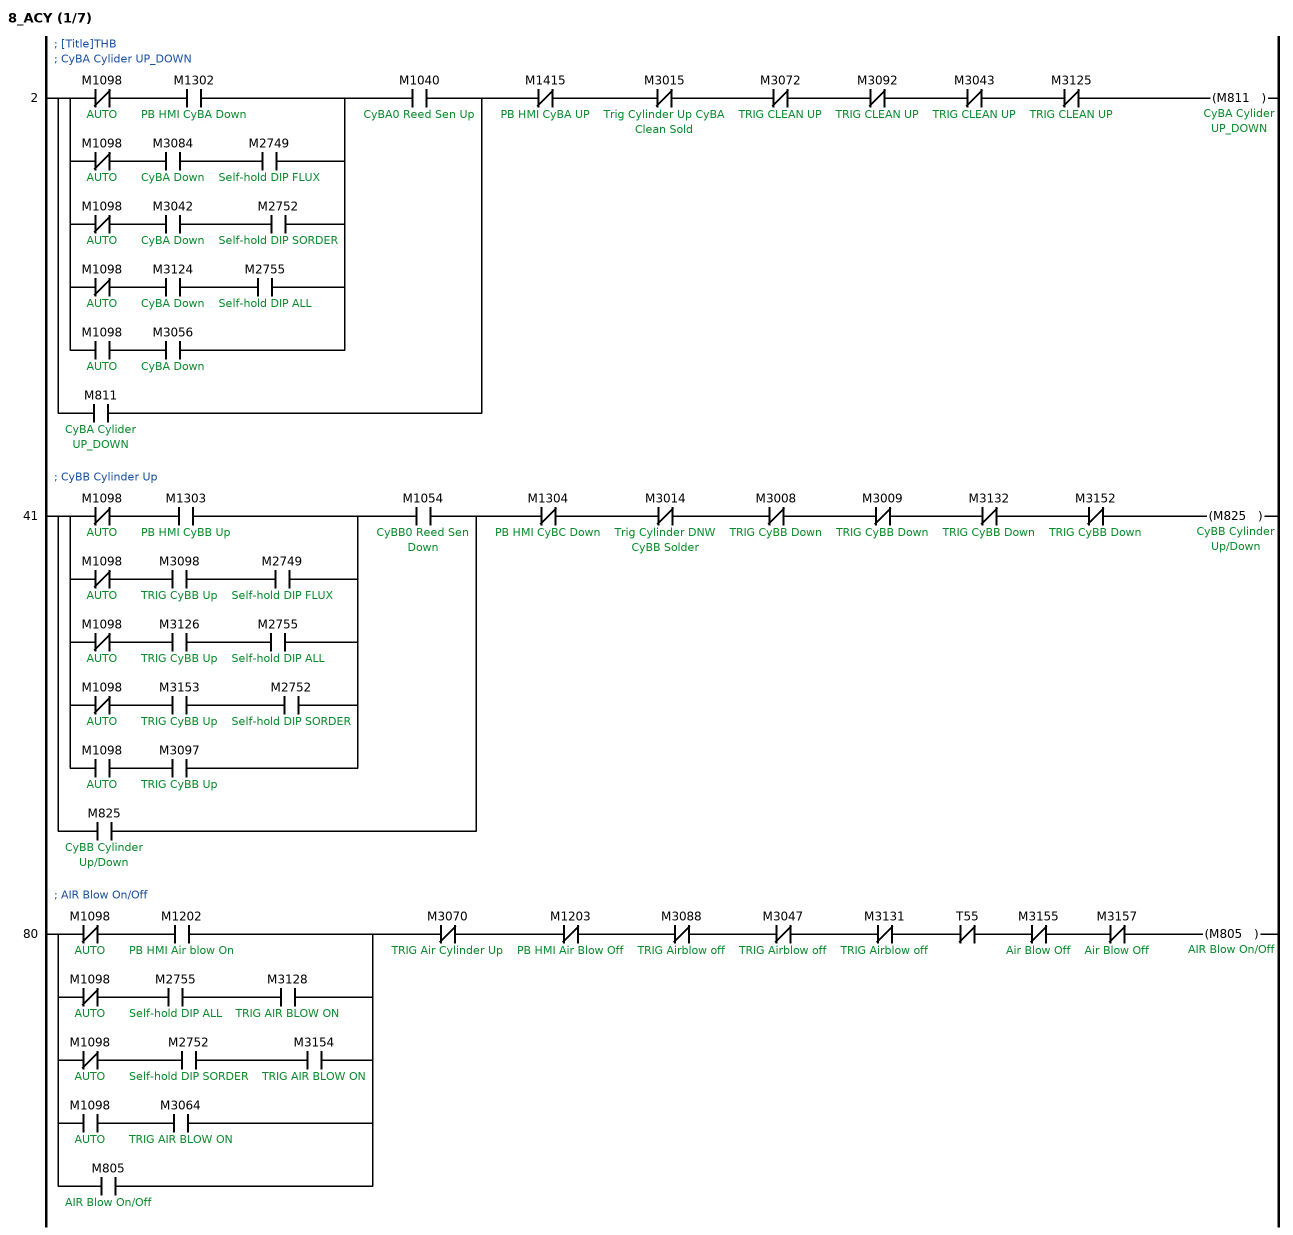
[picture p96: ladder of 8_ACY, rungs at steps 2 to 80]
; [Title]THB
; CyBA Cylider UP_DOWN
2     LDI     M1098  ; AUTO
      AND     M1302  ; PB HMI CyBA Down
      LDI     M1098  ; AUTO
      AND     M3084  ; CyBA Down
      AND     M2749  ; Self-hold DIP FLUX
      ORB
      LDI     M1098  ; AUTO
      AND     M3042  ; CyBA Down
      AND     M2752  ; Self-hold DIP SORDER
      ORB
      LDI     M1098  ; AUTO
      AND     M3124  ; CyBA Down
      AND     M2755  ; Self-hold DIP ALL
      ORB
      LD      M1098  ; AUTO
      AND     M3056  ; CyBA Down
      ORB
      AND     M1040  ; CyBA0 Reed Sen Up
      OR      M811  ; CyBA Cylider UP_DOWN
      ANI     M1415  ; PB HMI CyBA UP
      ANI     M3015  ; Trig Cylinder Up CyBA Clean Sold
      ANI     M3072  ; TRIG CLEAN UP
      ANI     M3092  ; TRIG CLEAN UP
      ANI     M3043  ; TRIG CLEAN UP
      ANI     M3125  ; TRIG CLEAN UP
      OUT     M811  ; CyBA Cylider UP_DOWN
; CyBB Cylinder Up
41    LDI     M1098  ; AUTO
      AND     M1303  ; PB HMI CyBB Up
      LDI     M1098  ; AUTO
      AND     M3098  ; TRIG CyBB Up
      AND     M2749  ; Self-hold DIP FLUX
      ORB
      LDI     M1098  ; AUTO
      AND     M3126  ; TRIG CyBB Up
      AND     M2755  ; Self-hold DIP ALL
      ORB
      LDI     M1098  ; AUTO
      AND     M3153  ; TRIG CyBB Up
      AND     M2752  ; Self-hold DIP SORDER
      ORB
      LD      M1098  ; AUTO
      AND     M3097  ; TRIG CyBB Up
      ORB
      AND     M1054  ; CyBB0 Reed Sen Down
      OR      M825  ; CyBB Cylinder Up/Down
      ANI     M1304  ; PB HMI CyBC Down
      ANI     M3014  ; Trig Cylinder DNW CyBB Solder
      ANI     M3008  ; TRIG CyBB Down
      ANI     M3009  ; TRIG CyBB Down
      ANI     M3132  ; TRIG CyBB Down
      ANI     M3152  ; TRIG CyBB Down
      OUT     M825  ; CyBB Cylinder Up/Down
; AIR Blow On/Off
80    LDI     M1098  ; AUTO
      AND     M1202  ; PB HMI Air blow On
      LDI     M1098  ; AUTO
      AND     M2755  ; Self-hold DIP ALL
      AND     M3128  ; TRIG AIR BLOW ON
      ORB
      LDI     M1098  ; AUTO
      AND     M2752  ; Self-hold DIP SORDER
      AND     M3154  ; TRIG AIR BLOW ON
      ORB
      LD      M1098  ; AUTO
      AND     M3064  ; TRIG AIR BLOW ON
      ORB
      OR      M805  ; AIR Blow On/Off
      ANI     M3070  ; TRIG Air Cylinder Up
      ANI     M1203  ; PB HMI Air Blow Off
      ANI     M3088  ; TRIG Airblow off
      ANI     M3047  ; TRIG Airblow off
      ANI     M3131  ; TRIG Airblow off
      ANI     T55
      ANI     M3155  ; Air Blow Off
      ANI     M3157  ; Air Blow Off
      OUT     M805  ; AIR Blow On/Off
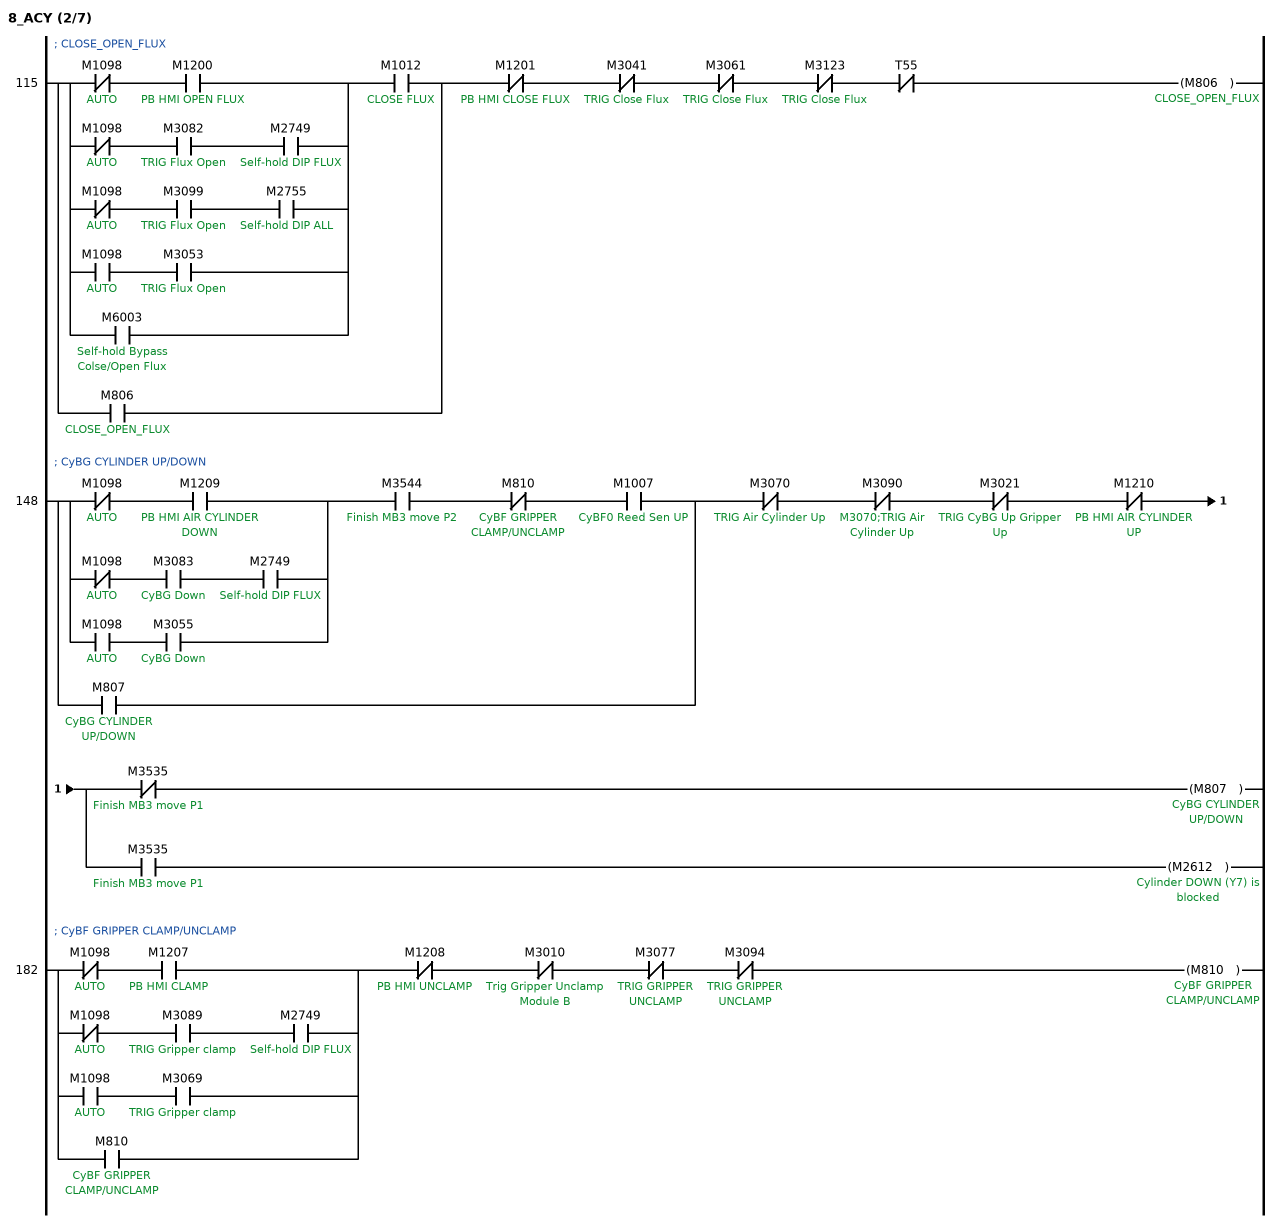
; CLOSE_OPEN_FLUX
115   LDI     M1098  ; AUTO
      AND     M1200  ; PB HMI OPEN FLUX
      LDI     M1098  ; AUTO
      AND     M3082  ; TRIG Flux Open
      AND     M2749  ; Self-hold DIP FLUX
      ORB
      LDI     M1098  ; AUTO
      AND     M3099  ; TRIG Flux Open
      AND     M2755  ; Self-hold DIP ALL
      ORB
      LD      M1098  ; AUTO
      AND     M3053  ; TRIG Flux Open
      ORB
      OR      M6003  ; Self-hold Bypass Colse/Open Flux
      AND     M1012  ; CLOSE FLUX
      OR      M806  ; CLOSE_OPEN_FLUX
      ANI     M1201  ; PB HMI CLOSE FLUX
      ANI     M3041  ; TRIG Close Flux
      ANI     M3061  ; TRIG Close Flux
      ANI     M3123  ; TRIG Close Flux
      ANI     T55
      OUT     M806  ; CLOSE_OPEN_FLUX
; CyBG CYLINDER UP/DOWN
148   LDI     M1098  ; AUTO
      AND     M1209  ; PB HMI AIR CYLINDER DOWN
      LDI     M1098  ; AUTO
      AND     M3083  ; CyBG Down
      AND     M2749  ; Self-hold DIP FLUX
      ORB
      LD      M1098  ; AUTO
      AND     M3055  ; CyBG Down
      ORB
      AND     M3544  ; Finish MB3 move P2
      ANI     M810  ; CyBF GRIPPER CLAMP/UNCLAMP
      AND     M1007  ; CyBF0 Reed Sen UP
      OR      M807  ; CyBG CYLINDER UP/DOWN
      ANI     M3070  ; TRIG Air Cylinder Up
      ANI     M3090  ; M3070;TRIG Air Cylinder Up
      ANI     M3021  ; TRIG CyBG Up Gripper Up
      ANI     M1210  ; PB HMI AIR CYLINDER UP
      MPS
      ANI     M3535  ; Finish MB3 move P1
      OUT     M807  ; CyBG CYLINDER UP/DOWN
      MPP
      AND     M3535  ; Finish MB3 move P1
      OUT     M2612  ; Cylinder DOWN (Y7) is blocked
; CyBF GRIPPER CLAMP/UNCLAMP
182   LDI     M1098  ; AUTO
      AND     M1207  ; PB HMI CLAMP
      LDI     M1098  ; AUTO
      AND     M3089  ; TRIG Gripper clamp
      AND     M2749  ; Self-hold DIP FLUX
      ORB
      LD      M1098  ; AUTO
      AND     M3069  ; TRIG Gripper clamp
      ORB
      OR      M810  ; CyBF GRIPPER CLAMP/UNCLAMP
      ANI     M1208  ; PB HMI UNCLAMP
      ANI     M3010  ; Trig Gripper Unclamp Module B
      ANI     M3077  ; TRIG GRIPPER UNCLAMP
      ANI     M3094  ; TRIG GRIPPER UNCLAMP
      OUT     M810  ; CyBF GRIPPER CLAMP/UNCLAMP
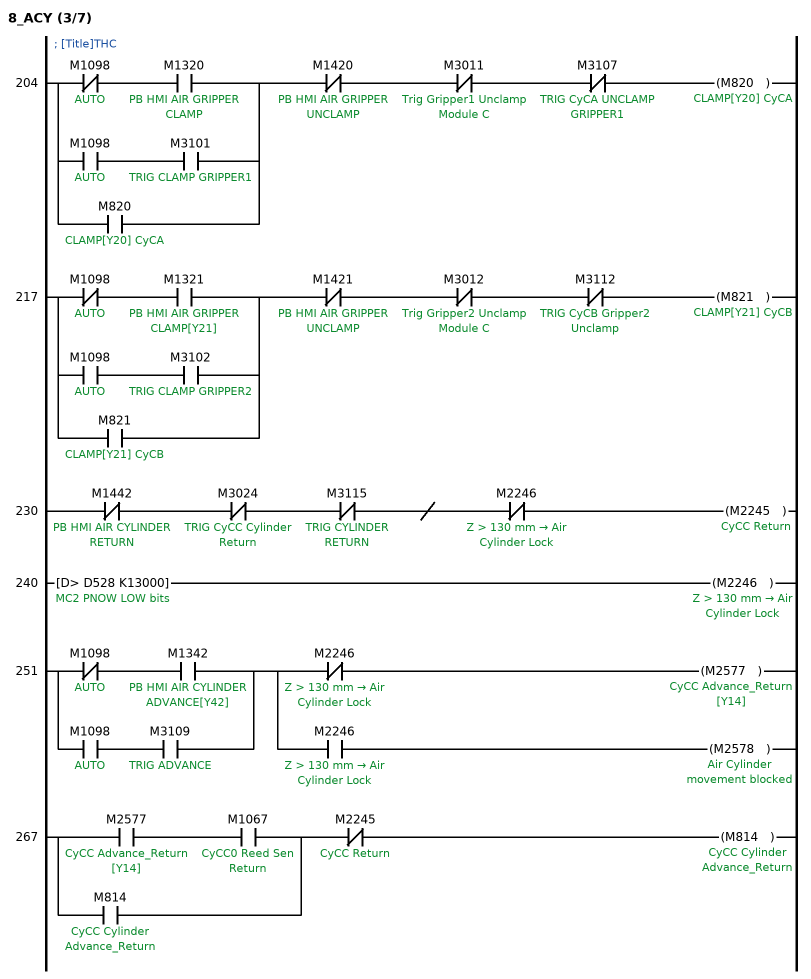
; [Title]THC
204   LDI     M1098  ; AUTO
      AND     M1320  ; PB HMI AIR GRIPPER CLAMP
      LD      M1098  ; AUTO
      AND     M3101  ; TRIG CLAMP GRIPPER1
      ORB
      OR      M820  ; CLAMP[Y20] CyCA
      ANI     M1420  ; PB HMI AIR GRIPPER UNCLAMP
      ANI     M3011  ; Trig Gripper1 Unclamp Module C
      ANI     M3107  ; TRIG CyCA UNCLAMP GRIPPER1
      OUT     M820  ; CLAMP[Y20] CyCA
217   LDI     M1098  ; AUTO
      AND     M1321  ; PB HMI AIR GRIPPER CLAMP[Y21]
      LD      M1098  ; AUTO
      AND     M3102  ; TRIG CLAMP GRIPPER2
      ORB
      OR      M821  ; CLAMP[Y21] CyCB
      ANI     M1421  ; PB HMI AIR GRIPPER UNCLAMP
      ANI     M3012  ; Trig Gripper2 Unclamp Module C
      ANI     M3112  ; TRIG CyCB Gripper2 Unclamp
      OUT     M821  ; CLAMP[Y21] CyCB
230   LDI     M1442  ; PB HMI AIR CYLINDER RETURN
      ANI     M3024  ; TRIG CyCC Cylinder Return
      ANI     M3115  ; TRIG CYLINDER RETURN
      INV
      ANI     M2246  ; Z > 130 mm → Air Cylinder Lock
      OUT     M2245  ; CyCC Return
240   LDD>    D528 K13000  ; MC2 PNOW LOW bits
      OUT     M2246  ; Z > 130 mm → Air Cylinder Lock
251   LDI     M1098  ; AUTO
      AND     M1342  ; PB HMI AIR CYLINDER ADVANCE[Y42]
      LD      M1098  ; AUTO
      AND     M3109  ; TRIG ADVANCE
      ORB
      MPS
      ANI     M2246  ; Z > 130 mm → Air Cylinder Lock
      OUT     M2577  ; CyCC Advance_Return [Y14]
      MPP
      AND     M2246  ; Z > 130 mm → Air Cylinder Lock
      OUT     M2578  ; Air Cylinder movement blocked
267   LD      M2577  ; CyCC Advance_Return [Y14]
      AND     M1067  ; CyCC0 Reed Sen Return
      OR      M814  ; CyCC Cylinder Advance_Return
      ANI     M2245  ; CyCC Return
      OUT     M814  ; CyCC Cylinder Advance_Return
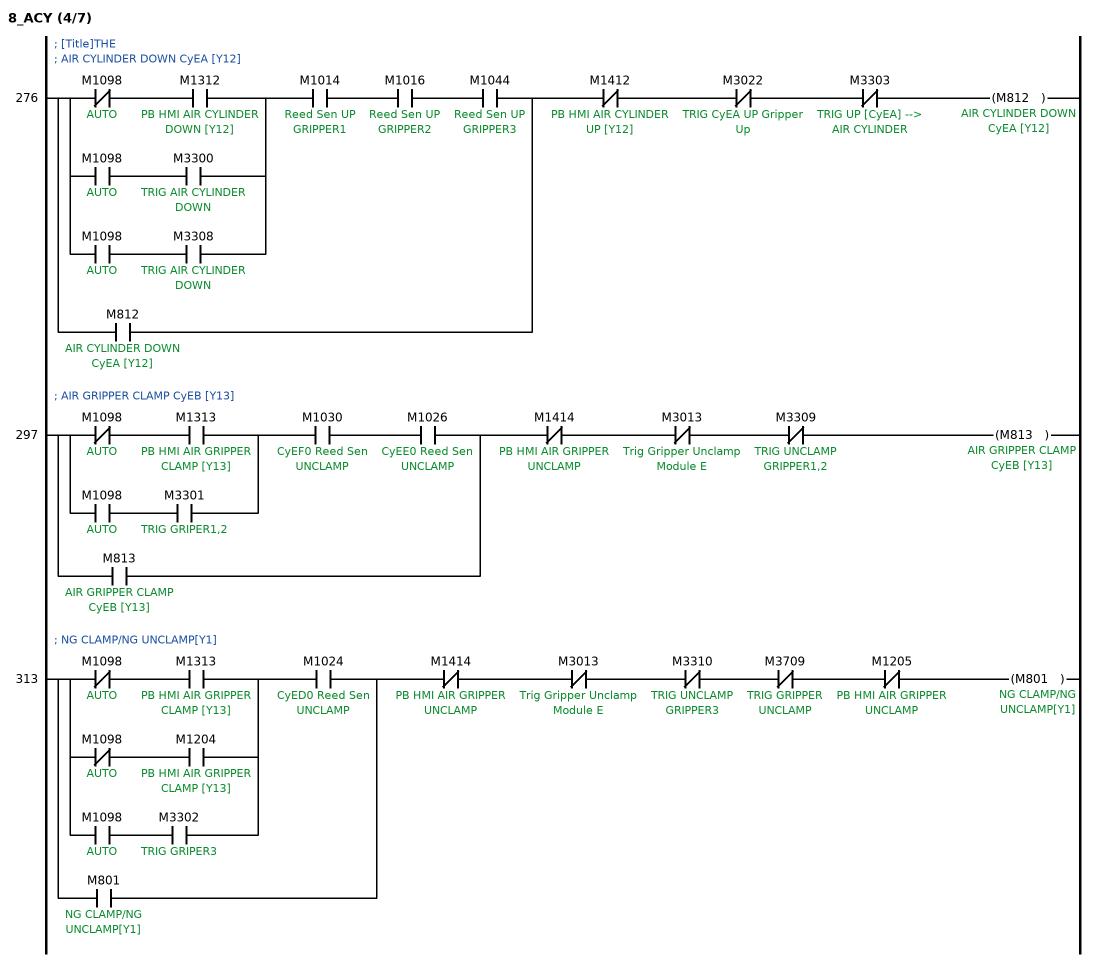
; [Title]THE
; AIR CYLINDER DOWN CyEA [Y12]
276   LDI     M1098  ; AUTO
      AND     M1312  ; PB HMI AIR CYLINDER DOWN [Y12]
      LD      M1098  ; AUTO
      AND     M3300  ; TRIG AIR CYLINDER DOWN
      ORB
      LD      M1098  ; AUTO
      AND     M3308  ; TRIG AIR CYLINDER DOWN
      ORB
      AND     M1014  ; Reed Sen UP GRIPPER1
      AND     M1016  ; Reed Sen UP GRIPPER2
      AND     M1044  ; Reed Sen UP GRIPPER3
      OR      M812  ; AIR CYLINDER DOWN CyEA [Y12]
      ANI     M1412  ; PB HMI AIR CYLINDER UP [Y12]
      ANI     M3022  ; TRIG CyEA UP Gripper Up
      ANI     M3303  ; TRIG UP [CyEA] --> AIR CYLINDER
      OUT     M812  ; AIR CYLINDER DOWN CyEA [Y12]
; AIR GRIPPER CLAMP CyEB [Y13]
297   LDI     M1098  ; AUTO
      AND     M1313  ; PB HMI AIR GRIPPER CLAMP [Y13]
      LD      M1098  ; AUTO
      AND     M3301  ; TRIG GRIPER1,2
      ORB
      AND     M1030  ; CyEF0 Reed Sen UNCLAMP
      AND     M1026  ; CyEE0 Reed Sen UNCLAMP
      OR      M813  ; AIR GRIPPER CLAMP CyEB [Y13]
      ANI     M1414  ; PB HMI AIR GRIPPER UNCLAMP
      ANI     M3013  ; Trig Gripper Unclamp Module E
      ANI     M3309  ; TRIG UNCLAMP GRIPPER1,2
      OUT     M813  ; AIR GRIPPER CLAMP CyEB [Y13]
; NG CLAMP/NG UNCLAMP[Y1]
313   LDI     M1098  ; AUTO
      AND     M1313  ; PB HMI AIR GRIPPER CLAMP [Y13]
      LDI     M1098  ; AUTO
      AND     M1204  ; PB HMI AIR GRIPPER CLAMP [Y13]
      ORB
      LD      M1098  ; AUTO
      AND     M3302  ; TRIG GRIPER3
      ORB
      AND     M1024  ; CyED0 Reed Sen UNCLAMP
      OR      M801  ; NG CLAMP/NG UNCLAMP[Y1]
      ANI     M1414  ; PB HMI AIR GRIPPER UNCLAMP
      ANI     M3013  ; Trig Gripper Unclamp Module E
      ANI     M3310  ; TRIG UNCLAMP GRIPPER3
      ANI     M3709  ; TRIG GRIPPER UNCLAMP
      ANI     M1205  ; PB HMI AIR GRIPPER UNCLAMP
      OUT     M801  ; NG CLAMP/NG UNCLAMP[Y1]
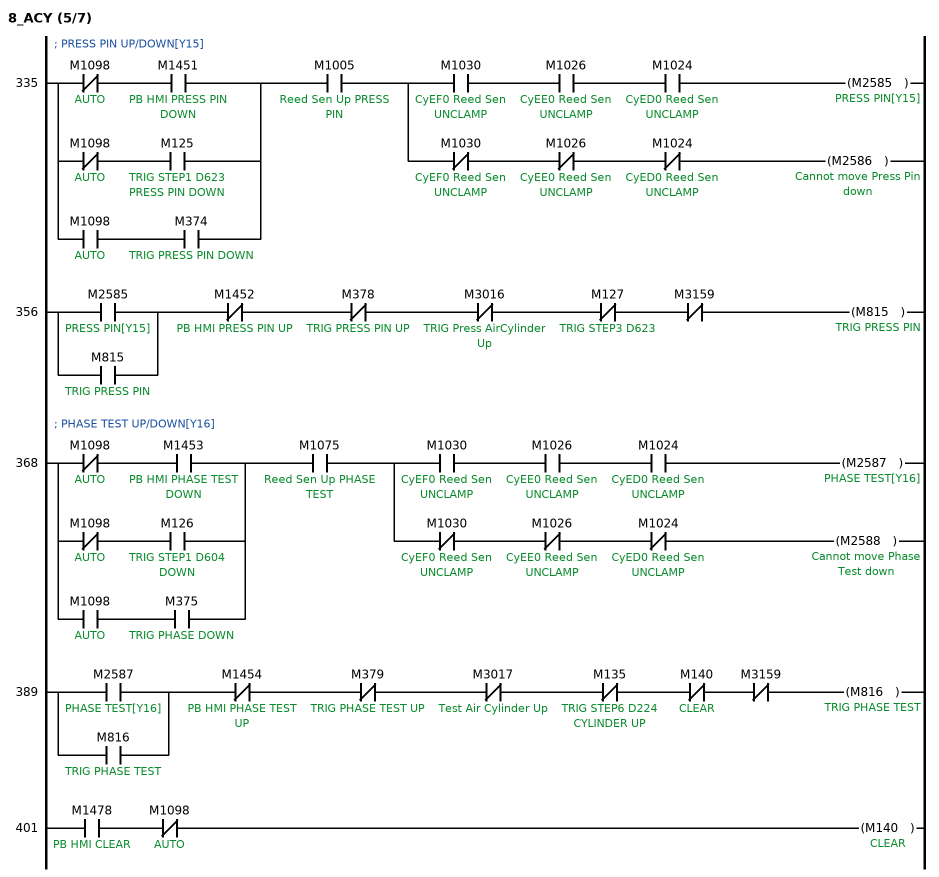
; PRESS PIN UP/DOWN[Y15]
335   LDI     M1098  ; AUTO
      AND     M1451  ; PB HMI PRESS PIN DOWN
      LDI     M1098  ; AUTO
      AND     M125  ; TRIG STEP1 D623 PRESS PIN DOWN
      ORB
      LD      M1098  ; AUTO
      AND     M374  ; TRIG PRESS PIN DOWN
      ORB
      AND     M1005  ; Reed Sen Up PRESS PIN
      MPS
      AND     M1030  ; CyEF0 Reed Sen UNCLAMP
      AND     M1026  ; CyEE0 Reed Sen UNCLAMP
      AND     M1024  ; CyED0 Reed Sen UNCLAMP
      OUT     M2585  ; PRESS PIN[Y15]
      MPP
      ANI     M1030  ; CyEF0 Reed Sen UNCLAMP
      ANI     M1026  ; CyEE0 Reed Sen UNCLAMP
      ANI     M1024  ; CyED0 Reed Sen UNCLAMP
      OUT     M2586  ; Cannot move Press Pin down
356   LD      M2585  ; PRESS PIN[Y15]
      OR      M815  ; TRIG PRESS PIN
      ANI     M1452  ; PB HMI PRESS PIN UP
      ANI     M378  ; TRIG PRESS PIN UP
      ANI     M3016  ; TRIG Press AirCylinder Up
      ANI     M127  ; TRIG STEP3 D623
      ANI     M3159
      OUT     M815  ; TRIG PRESS PIN
; PHASE TEST UP/DOWN[Y16]
368   LDI     M1098  ; AUTO
      AND     M1453  ; PB HMI PHASE TEST DOWN
      LDI     M1098  ; AUTO
      AND     M126  ; TRIG STEP1 D604 DOWN
      ORB
      LD      M1098  ; AUTO
      AND     M375  ; TRIG PHASE DOWN
      ORB
      AND     M1075  ; Reed Sen Up PHASE TEST
      MPS
      AND     M1030  ; CyEF0 Reed Sen UNCLAMP
      AND     M1026  ; CyEE0 Reed Sen UNCLAMP
      AND     M1024  ; CyED0 Reed Sen UNCLAMP
      OUT     M2587  ; PHASE TEST[Y16]
      MPP
      ANI     M1030  ; CyEF0 Reed Sen UNCLAMP
      ANI     M1026  ; CyEE0 Reed Sen UNCLAMP
      ANI     M1024  ; CyED0 Reed Sen UNCLAMP
      OUT     M2588  ; Cannot move Phase Test down
389   LD      M2587  ; PHASE TEST[Y16]
      OR      M816  ; TRIG PHASE TEST
      ANI     M1454  ; PB HMI PHASE TEST UP
      ANI     M379  ; TRIG PHASE TEST UP
      ANI     M3017  ; Test Air Cylinder Up
      ANI     M135  ; TRIG STEP6 D224 CYLINDER UP
      ANI     M140  ; CLEAR
      ANI     M3159
      OUT     M816  ; TRIG PHASE TEST
401   LD      M1478  ; PB HMI CLEAR
      ANI     M1098  ; AUTO
      OUT     M140  ; CLEAR
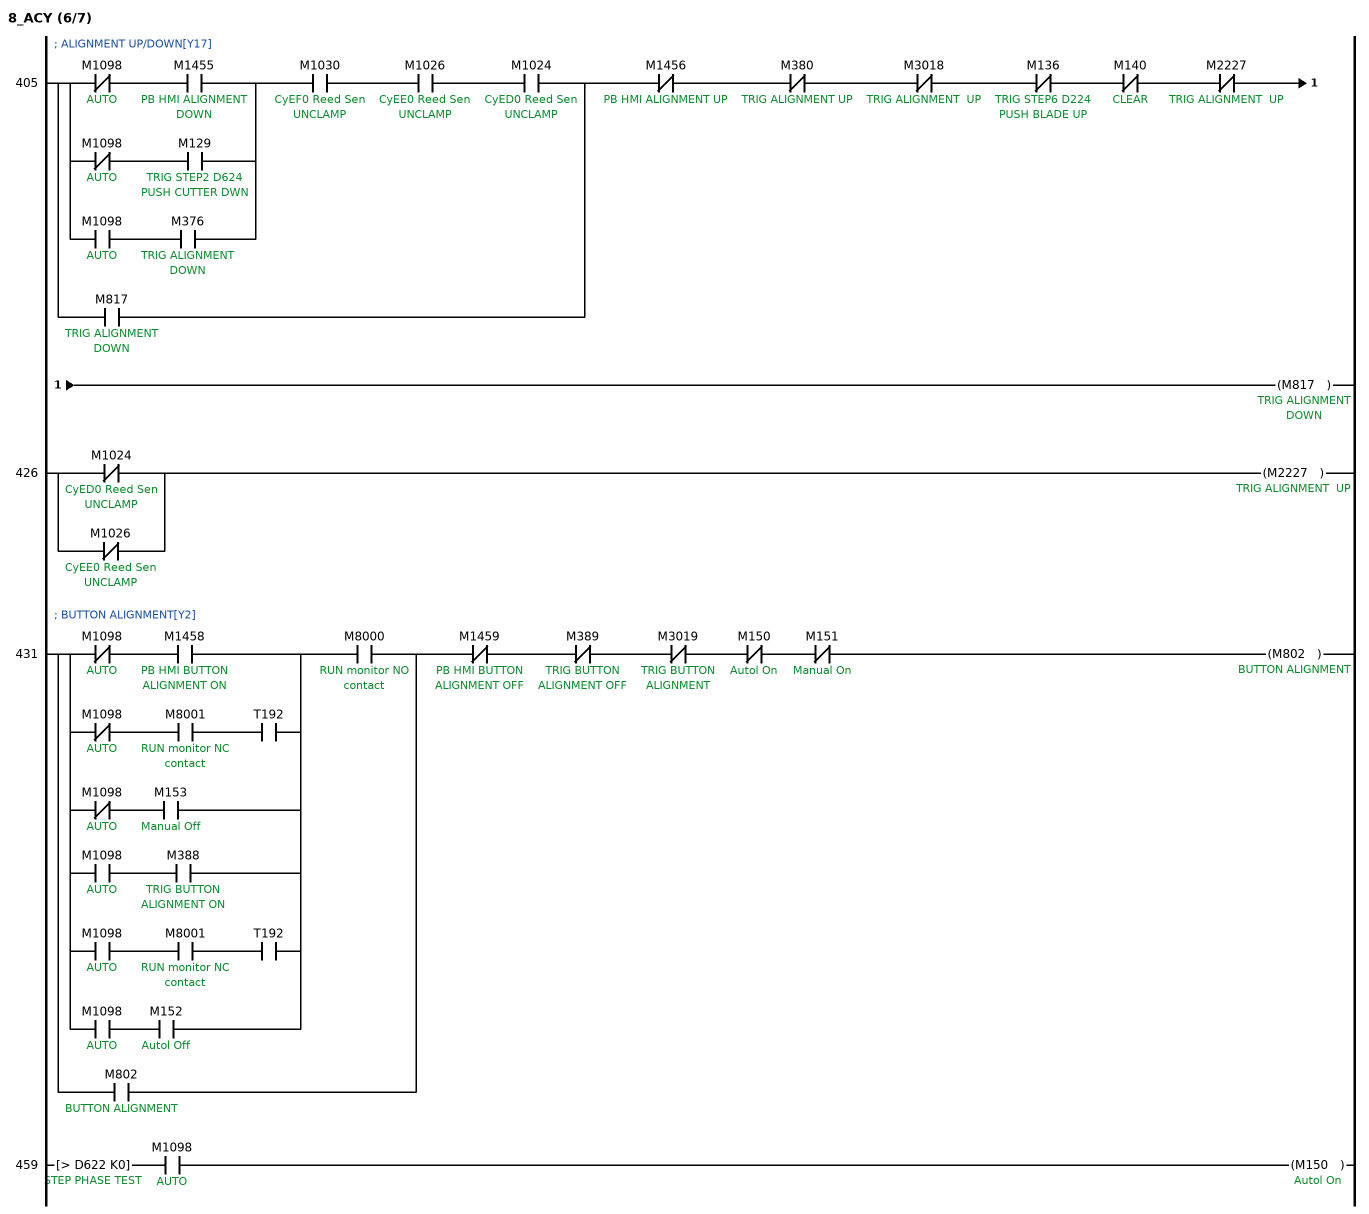
; ALIGNMENT UP/DOWN[Y17]
405   LDI     M1098  ; AUTO
      AND     M1455  ; PB HMI ALIGNMENT DOWN
      LDI     M1098  ; AUTO
      AND     M129  ; TRIG STEP2 D624 PUSH CUTTER DWN
      ORB
      LD      M1098  ; AUTO
      AND     M376  ; TRIG ALIGNMENT DOWN
      ORB
      AND     M1030  ; CyEF0 Reed Sen UNCLAMP
      AND     M1026  ; CyEE0 Reed Sen UNCLAMP
      AND     M1024  ; CyED0 Reed Sen UNCLAMP
      OR      M817  ; TRIG ALIGNMENT  DOWN
      ANI     M1456  ; PB HMI ALIGNMENT UP
      ANI     M380  ; TRIG ALIGNMENT UP
      ANI     M3018  ; TRIG ALIGNMENT  UP
      ANI     M136  ; TRIG STEP6 D224 PUSH BLADE UP
      ANI     M140  ; CLEAR
      ANI     M2227  ; TRIG ALIGNMENT  UP
      OUT     M817  ; TRIG ALIGNMENT  DOWN
426   LDI     M1024  ; CyED0 Reed Sen UNCLAMP
      ORI     M1026  ; CyEE0 Reed Sen UNCLAMP
      OUT     M2227  ; TRIG ALIGNMENT  UP
; BUTTON ALIGNMENT[Y2]
431   LDI     M1098  ; AUTO
      AND     M1458  ; PB HMI BUTTON ALIGNMENT ON
      LDI     M1098  ; AUTO
      AND     M8001  ; RUN monitor NC contact
      AND     T192
      ORB
      LDI     M1098  ; AUTO
      AND     M153  ; Manual Off
      ORB
      LD      M1098  ; AUTO
      AND     M388  ; TRIG BUTTON ALIGNMENT ON
      ORB
      LD      M1098  ; AUTO
      AND     M8001  ; RUN monitor NC contact
      AND     T192
      ORB
      LD      M1098  ; AUTO
      AND     M152  ; Autol Off
      ORB
      AND     M8000  ; RUN monitor NO contact
      OR      M802  ; BUTTON ALIGNMENT
      ANI     M1459  ; PB HMI BUTTON ALIGNMENT OFF
      ANI     M389  ; TRIG BUTTON ALIGNMENT OFF
      ANI     M3019  ; TRIG BUTTON ALIGNMENT
      ANI     M150  ; Autol On
      ANI     M151  ; Manual On
      OUT     M802  ; BUTTON ALIGNMENT
459   LD>     D622 K0  ; STEP PHASE TEST
      AND     M1098  ; AUTO
      OUT     M150  ; Autol On
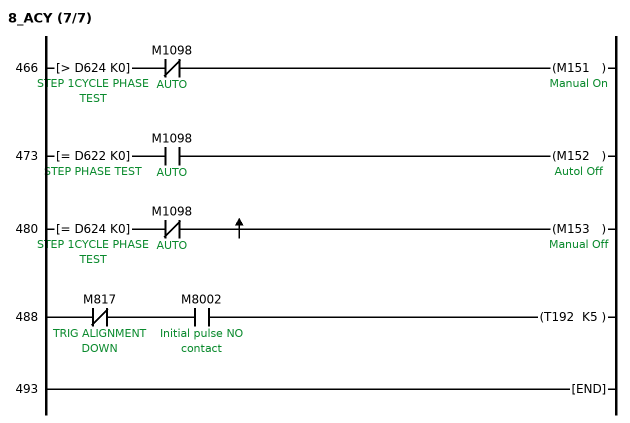
466   LD>     D624 K0  ; STEP 1CYCLE PHASE TEST
      ANI     M1098  ; AUTO
      OUT     M151  ; Manual On
473   LD=     D622 K0  ; STEP PHASE TEST
      AND     M1098  ; AUTO
      OUT     M152  ; Autol Off
480   LD=     D624 K0  ; STEP 1CYCLE PHASE TEST
      ANI     M1098  ; AUTO
      MEP
      OUT     M153  ; Manual Off
488   LDI     M817  ; TRIG ALIGNMENT  DOWN
      AND     M8002  ; Initial pulse NO contact
      OUT     T192 K5
493   END
END_PROGRAM

PROGRAM 90_IAI
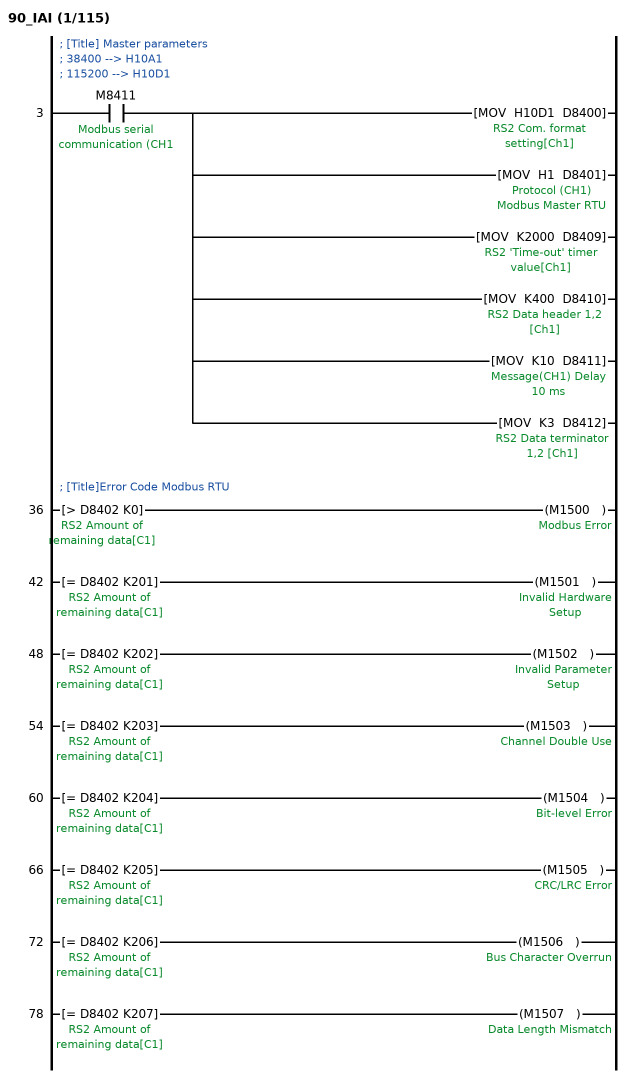
; [Title] Master parameters
; 38400 --> H10A1
; 115200 --> H10D1
3     LD      M8411  ; Modbus serial communication (CH1
      MOV     H10D1 D8400  ; RS2 Com. format setting[Ch1]
      MOV     H1 D8401  ; Protocol (CH1) Modbus Master RTU
      MOV     K2000 D8409  ; RS2 'Time-out' timer value[Ch1]
      MOV     K400 D8410  ; RS2 Data header 1,2 [Ch1]
      MOV     K10 D8411  ; Message(CH1) Delay 10 ms
      MOV     K3 D8412  ; RS2 Data terminator 1,2 [Ch1]
; [Title]Error Code Modbus RTU
36    LD>     D8402 K0  ; RS2 Amount of remaining data[C1]
      OUT     M1500  ; Modbus Error
42    LD=     D8402 K201  ; RS2 Amount of remaining data[C1]
      OUT     M1501  ; Invalid Hardware Setup
48    LD=     D8402 K202  ; RS2 Amount of remaining data[C1]
      OUT     M1502  ; Invalid Parameter Setup
54    LD=     D8402 K203  ; RS2 Amount of remaining data[C1]
      OUT     M1503  ; Channel Double Use
60    LD=     D8402 K204  ; RS2 Amount of remaining data[C1]
      OUT     M1504  ; Bit-level Error
66    LD=     D8402 K205  ; RS2 Amount of remaining data[C1]
      OUT     M1505  ; CRC/LRC Error
72    LD=     D8402 K206  ; RS2 Amount of remaining data[C1]
      OUT     M1506  ; Bus Character Overrun
78    LD=     D8402 K207  ; RS2 Amount of remaining data[C1]
      OUT     M1507  ; Data Length Mismatch
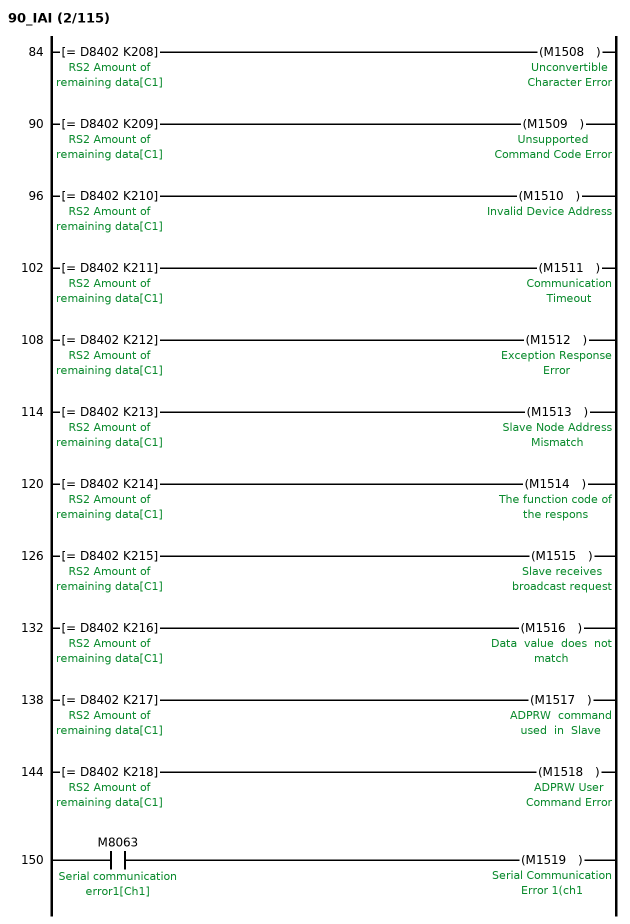
84    LD=     D8402 K208  ; RS2 Amount of remaining data[C1]
      OUT     M1508  ; Unconvertible Character Error
90    LD=     D8402 K209  ; RS2 Amount of remaining data[C1]
      OUT     M1509  ; Unsupported Command Code Error
96    LD=     D8402 K210  ; RS2 Amount of remaining data[C1]
      OUT     M1510  ; Invalid Device Address
102   LD=     D8402 K211  ; RS2 Amount of remaining data[C1]
      OUT     M1511  ; Communication Timeout
108   LD=     D8402 K212  ; RS2 Amount of remaining data[C1]
      OUT     M1512  ; Exception Response Error
114   LD=     D8402 K213  ; RS2 Amount of remaining data[C1]
      OUT     M1513  ; Slave Node Address Mismatch
120   LD=     D8402 K214  ; RS2 Amount of remaining data[C1]
      OUT     M1514  ; The function code of the respons
126   LD=     D8402 K215  ; RS2 Amount of remaining data[C1]
      OUT     M1515  ; Slave receives broadcast request
132   LD=     D8402 K216  ; RS2 Amount of remaining data[C1]
      OUT     M1516  ; Data  value  does  not  match
138   LD=     D8402 K217  ; RS2 Amount of remaining data[C1]
      OUT     M1517  ; ADPRW  command  used  in  Slave
144   LD=     D8402 K218  ; RS2 Amount of remaining data[C1]
      OUT     M1518  ; ADPRW User Command Error
150   LD      M8063  ; Serial communication error1[Ch1]
      OUT     M1519  ; Serial Communication Error 1(ch1
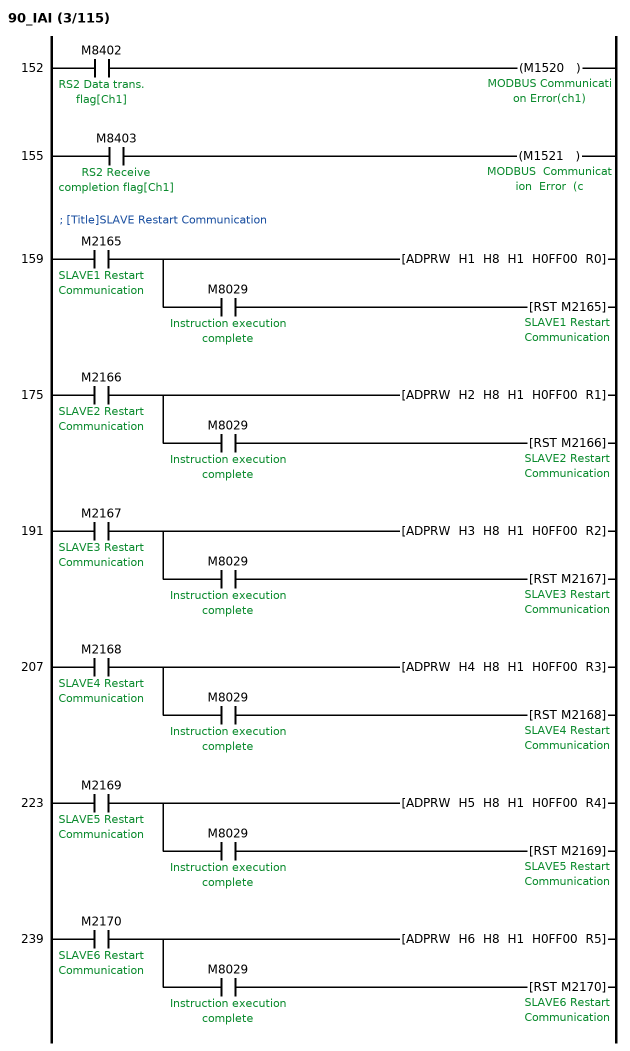
152   LD      M8402  ; RS2 Data trans. flag[Ch1]
      OUT     M1520  ; MODBUS Communication Error(ch1)
155   LD      M8403  ; RS2 Receive completion flag[Ch1]
      OUT     M1521  ; MODBUS  Communication  Error  (c
; [Title]SLAVE Restart Communication
159   LD      M2165  ; SLAVE1 Restart Communication
      ADPRW   H1 H8 H1 H0FF00 R0
      AND     M8029  ; Instruction execution complete
      RST     M2165  ; SLAVE1 Restart Communication
175   LD      M2166  ; SLAVE2 Restart Communication
      ADPRW   H2 H8 H1 H0FF00 R1
      AND     M8029  ; Instruction execution complete
      RST     M2166  ; SLAVE2 Restart Communication
191   LD      M2167  ; SLAVE3 Restart Communication
      ADPRW   H3 H8 H1 H0FF00 R2
      AND     M8029  ; Instruction execution complete
      RST     M2167  ; SLAVE3 Restart Communication
207   LD      M2168  ; SLAVE4 Restart Communication
      ADPRW   H4 H8 H1 H0FF00 R3
      AND     M8029  ; Instruction execution complete
      RST     M2168  ; SLAVE4 Restart Communication
223   LD      M2169  ; SLAVE5 Restart Communication
      ADPRW   H5 H8 H1 H0FF00 R4
      AND     M8029  ; Instruction execution complete
      RST     M2169  ; SLAVE5 Restart Communication
239   LD      M2170  ; SLAVE6 Restart Communication
      ADPRW   H6 H8 H1 H0FF00 R5
      AND     M8029  ; Instruction execution complete
      RST     M2170  ; SLAVE6 Restart Communication
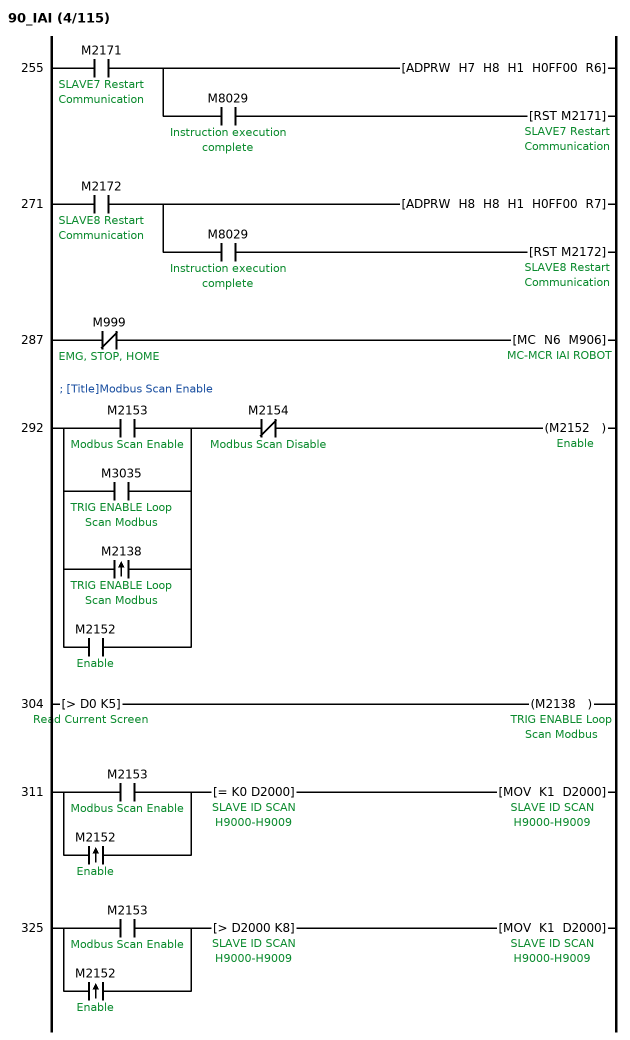
255   LD      M2171  ; SLAVE7 Restart Communication
      ADPRW   H7 H8 H1 H0FF00 R6
      AND     M8029  ; Instruction execution complete
      RST     M2171  ; SLAVE7 Restart Communication
271   LD      M2172  ; SLAVE8 Restart Communication
      ADPRW   H8 H8 H1 H0FF00 R7
      AND     M8029  ; Instruction execution complete
      RST     M2172  ; SLAVE8 Restart Communication
287   LDI     M999  ; EMG, STOP, HOME
      MC      N6 M906  ; MC-MCR IAI ROBOT
; [Title]Modbus Scan Enable
292   LD      M2153  ; Modbus Scan Enable
      OR      M3035  ; TRIG ENABLE Loop Scan Modbus
      ORP     M2138  ; TRIG ENABLE Loop Scan Modbus
      OR      M2152  ; Enable
      ANI     M2154  ; Modbus Scan Disable
      OUT     M2152  ; Enable
304   LD>     D0 K5  ; Read Current Screen
      OUT     M2138  ; TRIG ENABLE Loop Scan Modbus
311   LD      M2153  ; Modbus Scan Enable
      ORP     M2152  ; Enable
      AND=    K0 D2000  ; SLAVE ID SCAN H9000-H9009
      MOV     K1 D2000
325   LD      M2153  ; Modbus Scan Enable
      ORP     M2152  ; Enable
      AND>    D2000 K8  ; SLAVE ID SCAN H9000-H9009
      MOV     K1 D2000
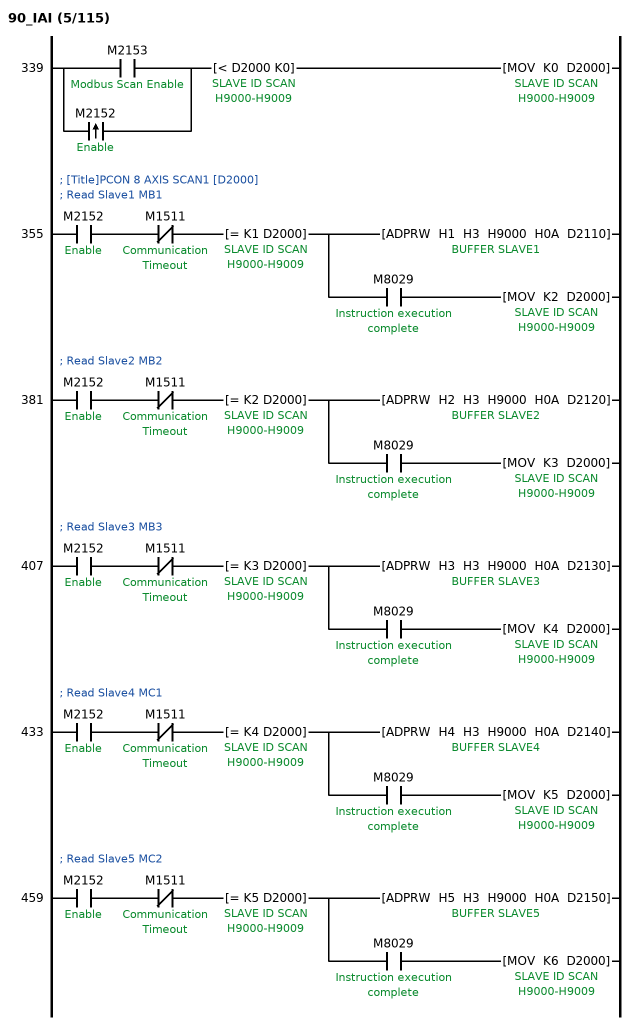
339   LD      M2153  ; Modbus Scan Enable
      ORP     M2152  ; Enable
      AND<    D2000 K0  ; SLAVE ID SCAN H9000-H9009
      MOV     K0 D2000
; [Title]PCON 8 AXIS SCAN1 [D2000]
; Read Slave1 MB1
355   LD      M2152  ; Enable
      ANI     M1511  ; Communication Timeout
      AND=    K1 D2000  ; SLAVE ID SCAN H9000-H9009
      ADPRW   H1 H3 H9000 H0A D2110  ; BUFFER SLAVE1
      AND     M8029  ; Instruction execution complete
      MOV     K2 D2000
; Read Slave2 MB2
381   LD      M2152  ; Enable
      ANI     M1511  ; Communication Timeout
      AND=    K2 D2000  ; SLAVE ID SCAN H9000-H9009
      ADPRW   H2 H3 H9000 H0A D2120  ; BUFFER SLAVE2
      AND     M8029  ; Instruction execution complete
      MOV     K3 D2000
; Read Slave3 MB3
407   LD      M2152  ; Enable
      ANI     M1511  ; Communication Timeout
      AND=    K3 D2000  ; SLAVE ID SCAN H9000-H9009
      ADPRW   H3 H3 H9000 H0A D2130  ; BUFFER SLAVE3
      AND     M8029  ; Instruction execution complete
      MOV     K4 D2000
; Read Slave4 MC1
433   LD      M2152  ; Enable
      ANI     M1511  ; Communication Timeout
      AND=    K4 D2000  ; SLAVE ID SCAN H9000-H9009
      ADPRW   H4 H3 H9000 H0A D2140  ; BUFFER SLAVE4
      AND     M8029  ; Instruction execution complete
      MOV     K5 D2000
; Read Slave5 MC2
459   LD      M2152  ; Enable
      ANI     M1511  ; Communication Timeout
      AND=    K5 D2000  ; SLAVE ID SCAN H9000-H9009
      ADPRW   H5 H3 H9000 H0A D2150  ; BUFFER SLAVE5
      AND     M8029  ; Instruction execution complete
      MOV     K6 D2000
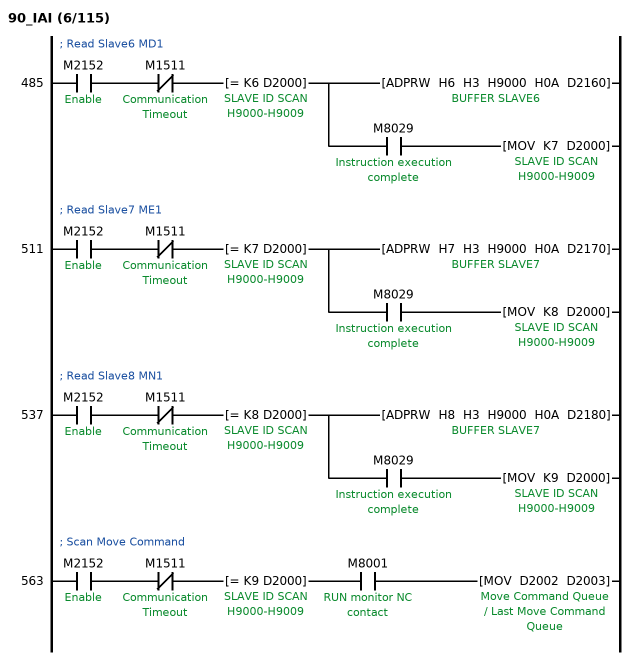
; Read Slave6 MD1
485   LD      M2152  ; Enable
      ANI     M1511  ; Communication Timeout
      AND=    K6 D2000  ; SLAVE ID SCAN H9000-H9009
      ADPRW   H6 H3 H9000 H0A D2160  ; BUFFER SLAVE6
      AND     M8029  ; Instruction execution complete
      MOV     K7 D2000
; Read Slave7 ME1
511   LD      M2152  ; Enable
      ANI     M1511  ; Communication Timeout
      AND=    K7 D2000  ; SLAVE ID SCAN H9000-H9009
      ADPRW   H7 H3 H9000 H0A D2170  ; BUFFER SLAVE7
      AND     M8029  ; Instruction execution complete
      MOV     K8 D2000
; Read Slave8 MN1
537   LD      M2152  ; Enable
      ANI     M1511  ; Communication Timeout
      AND=    K8 D2000  ; SLAVE ID SCAN H9000-H9009
      ADPRW   H8 H3 H9000 H0A D2180  ; BUFFER SLAVE7
      AND     M8029  ; Instruction execution complete
      MOV     K9 D2000
; Scan Move Command
563   LD      M2152  ; Enable
      ANI     M1511  ; Communication Timeout
      AND=    K9 D2000  ; SLAVE ID SCAN H9000-H9009
      AND     M8001  ; RUN monitor NC contact
      MOV     D2002 D2003  ; Move Command Queue / Last Move Command Queue
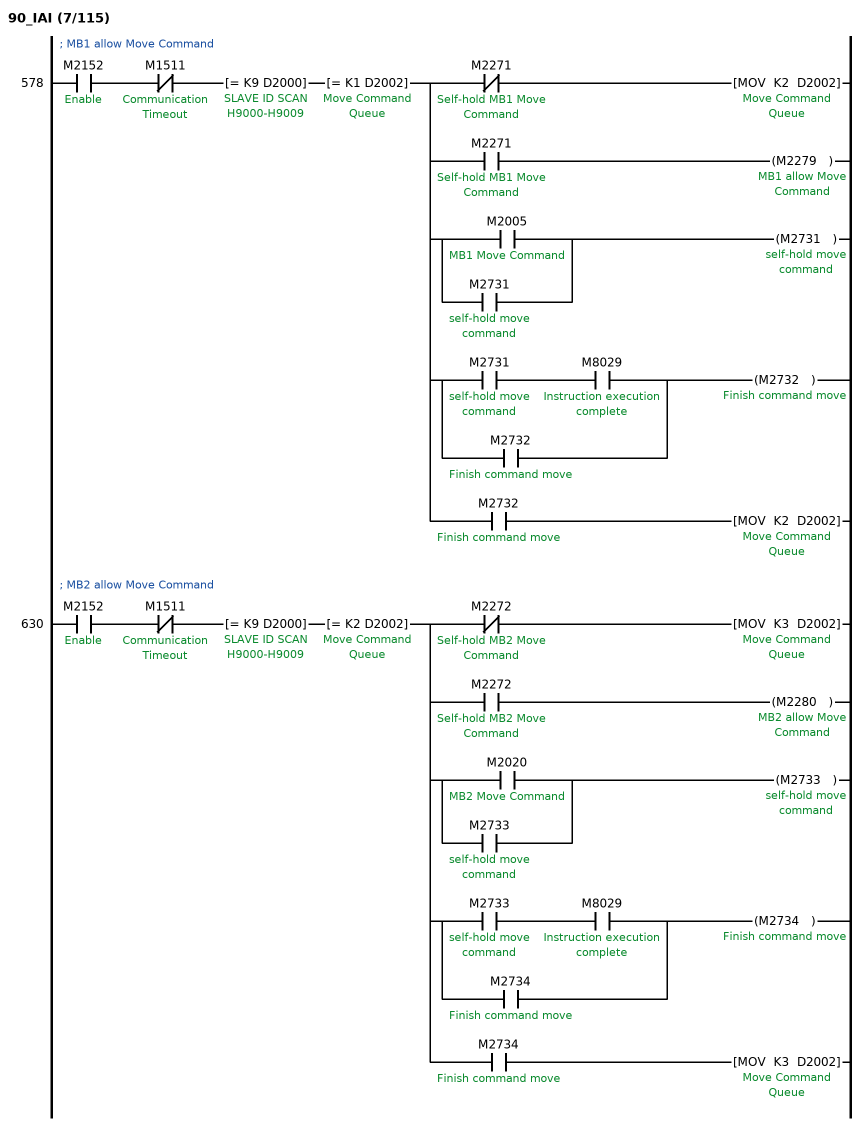
; MB1 allow Move Command
578   LD      M2152  ; Enable
      ANI     M1511  ; Communication Timeout
      AND=    K9 D2000  ; SLAVE ID SCAN H9000-H9009
      AND=    K1 D2002  ; Move Command Queue
      MPS
      ANI     M2271  ; Self-hold MB1 Move Command
      MOV     K2 D2002
      MRD
      AND     M2271  ; Self-hold MB1 Move Command
      OUT     M2279  ; MB1 allow Move Command
      MRD
      LD      M2005  ; MB1 Move Command
      OR      M2731  ; self-hold move command
      ANB
      OUT     M2731  ; self-hold move command
      MRD
      LD      M2731  ; self-hold move command
      AND     M8029  ; Instruction execution complete
      OR      M2732  ; Finish command move
      ANB
      OUT     M2732  ; Finish command move
      MPP
      AND     M2732  ; Finish command move
      MOV     K2 D2002
; MB2 allow Move Command
630   LD      M2152  ; Enable
      ANI     M1511  ; Communication Timeout
      AND=    K9 D2000  ; SLAVE ID SCAN H9000-H9009
      AND=    K2 D2002  ; Move Command Queue
      MPS
      ANI     M2272  ; Self-hold MB2 Move Command
      MOV     K3 D2002
      MRD
      AND     M2272  ; Self-hold MB2 Move Command
      OUT     M2280  ; MB2 allow Move Command
      MRD
      LD      M2020  ; MB2 Move Command
      OR      M2733  ; self-hold move command
      ANB
      OUT     M2733  ; self-hold move command
      MRD
      LD      M2733  ; self-hold move command
      AND     M8029  ; Instruction execution complete
      OR      M2734  ; Finish command move
      ANB
      OUT     M2734  ; Finish command move
      MPP
      AND     M2734  ; Finish command move
      MOV     K3 D2002
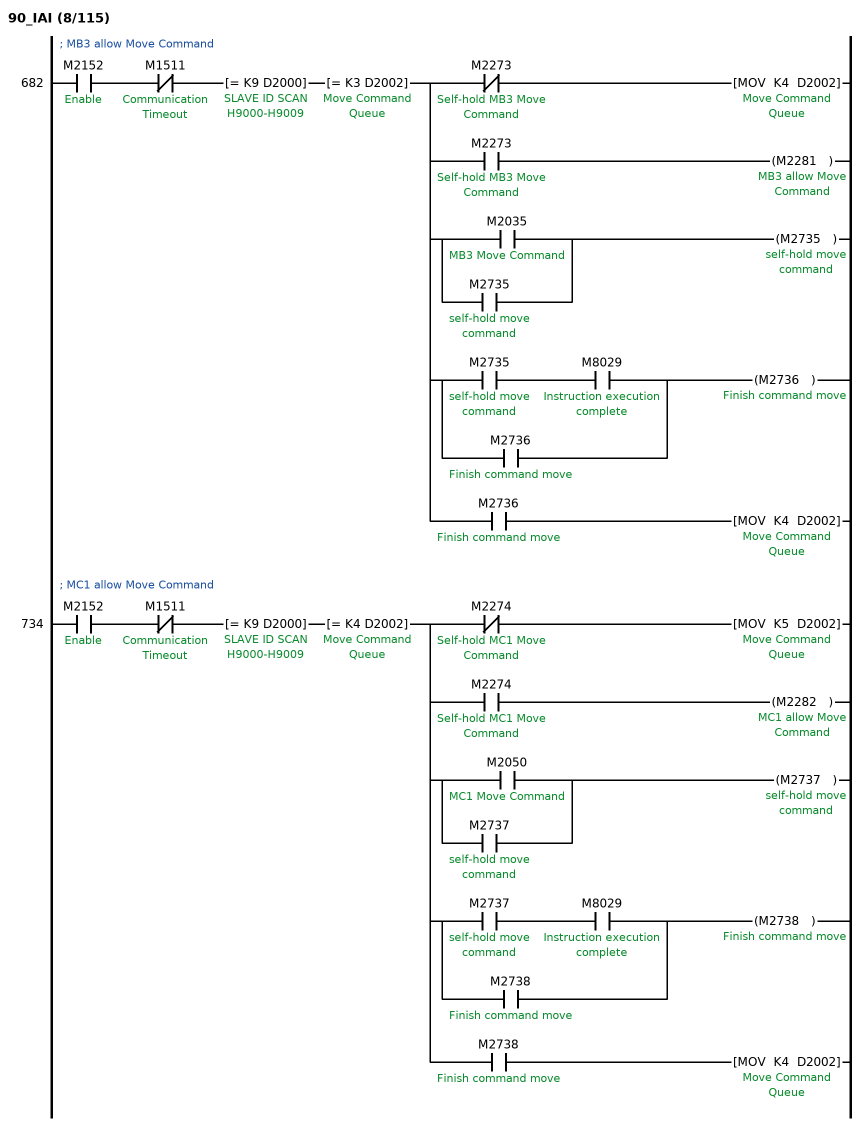
; MB3 allow Move Command
682   LD      M2152  ; Enable
      ANI     M1511  ; Communication Timeout
      AND=    K9 D2000  ; SLAVE ID SCAN H9000-H9009
      AND=    K3 D2002  ; Move Command Queue
      MPS
      ANI     M2273  ; Self-hold MB3 Move Command
      MOV     K4 D2002
      MRD
      AND     M2273  ; Self-hold MB3 Move Command
      OUT     M2281  ; MB3 allow Move Command
      MRD
      LD      M2035  ; MB3 Move Command
      OR      M2735  ; self-hold move command
      ANB
      OUT     M2735  ; self-hold move command
      MRD
      LD      M2735  ; self-hold move command
      AND     M8029  ; Instruction execution complete
      OR      M2736  ; Finish command move
      ANB
      OUT     M2736  ; Finish command move
      MPP
      AND     M2736  ; Finish command move
      MOV     K4 D2002
; MC1 allow Move Command
734   LD      M2152  ; Enable
      ANI     M1511  ; Communication Timeout
      AND=    K9 D2000  ; SLAVE ID SCAN H9000-H9009
      AND=    K4 D2002  ; Move Command Queue
      MPS
      ANI     M2274  ; Self-hold MC1 Move Command
      MOV     K5 D2002
      MRD
      AND     M2274  ; Self-hold MC1 Move Command
      OUT     M2282  ; MC1 allow Move Command
      MRD
      LD      M2050  ; MC1 Move Command
      OR      M2737  ; self-hold move command
      ANB
      OUT     M2737  ; self-hold move command
      MRD
      LD      M2737  ; self-hold move command
      AND     M8029  ; Instruction execution complete
      OR      M2738  ; Finish command move
      ANB
      OUT     M2738  ; Finish command move
      MPP
      AND     M2738  ; Finish command move
      MOV     K4 D2002
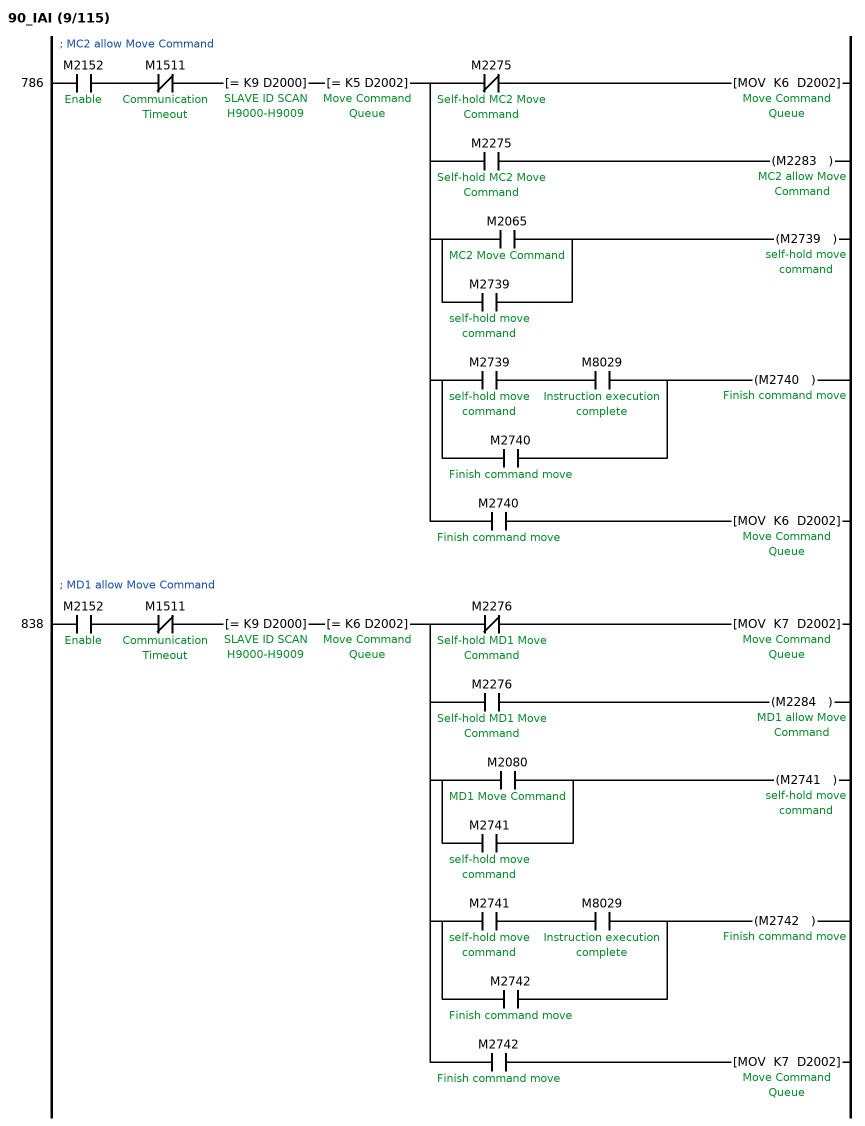
; MC2 allow Move Command
786   LD      M2152  ; Enable
      ANI     M1511  ; Communication Timeout
      AND=    K9 D2000  ; SLAVE ID SCAN H9000-H9009
      AND=    K5 D2002  ; Move Command Queue
      MPS
      ANI     M2275  ; Self-hold MC2 Move Command
      MOV     K6 D2002
      MRD
      AND     M2275  ; Self-hold MC2 Move Command
      OUT     M2283  ; MC2 allow Move Command
      MRD
      LD      M2065  ; MC2 Move Command
      OR      M2739  ; self-hold move command
      ANB
      OUT     M2739  ; self-hold move command
      MRD
      LD      M2739  ; self-hold move command
      AND     M8029  ; Instruction execution complete
      OR      M2740  ; Finish command move
      ANB
      OUT     M2740  ; Finish command move
      MPP
      AND     M2740  ; Finish command move
      MOV     K6 D2002
; MD1 allow Move Command
838   LD      M2152  ; Enable
      ANI     M1511  ; Communication Timeout
      AND=    K9 D2000  ; SLAVE ID SCAN H9000-H9009
      AND=    K6 D2002  ; Move Command Queue
      MPS
      ANI     M2276  ; Self-hold MD1 Move Command
      MOV     K7 D2002
      MRD
      AND     M2276  ; Self-hold MD1 Move Command
      OUT     M2284  ; MD1 allow Move Command
      MRD
      LD      M2080  ; MD1 Move Command
      OR      M2741  ; self-hold move command
      ANB
      OUT     M2741  ; self-hold move command
      MRD
      LD      M2741  ; self-hold move command
      AND     M8029  ; Instruction execution complete
      OR      M2742  ; Finish command move
      ANB
      OUT     M2742  ; Finish command move
      MPP
      AND     M2742  ; Finish command move
      MOV     K7 D2002
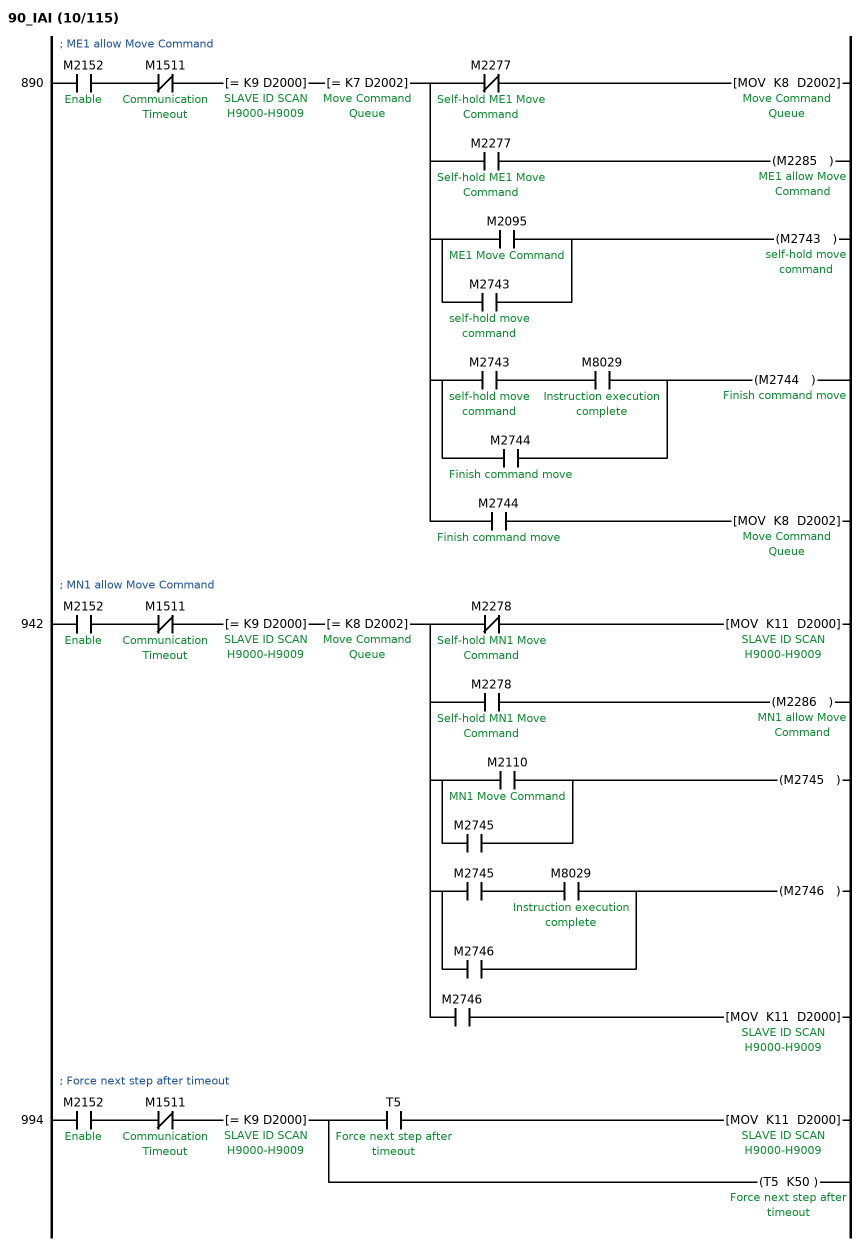
; ME1 allow Move Command
890   LD      M2152  ; Enable
      ANI     M1511  ; Communication Timeout
      AND=    K9 D2000  ; SLAVE ID SCAN H9000-H9009
      AND=    K7 D2002  ; Move Command Queue
      MPS
      ANI     M2277  ; Self-hold ME1 Move Command
      MOV     K8 D2002
      MRD
      AND     M2277  ; Self-hold ME1 Move Command
      OUT     M2285  ; ME1 allow Move Command
      MRD
      LD      M2095  ; ME1 Move Command
      OR      M2743  ; self-hold move command
      ANB
      OUT     M2743  ; self-hold move command
      MRD
      LD      M2743  ; self-hold move command
      AND     M8029  ; Instruction execution complete
      OR      M2744  ; Finish command move
      ANB
      OUT     M2744  ; Finish command move
      MPP
      AND     M2744  ; Finish command move
      MOV     K8 D2002
; MN1 allow Move Command
942   LD      M2152  ; Enable
      ANI     M1511  ; Communication Timeout
      AND=    K9 D2000  ; SLAVE ID SCAN H9000-H9009
      AND=    K8 D2002  ; Move Command Queue
      MPS
      ANI     M2278  ; Self-hold MN1 Move Command
      MOV     K11 D2000
      MRD
      AND     M2278  ; Self-hold MN1 Move Command
      OUT     M2286  ; MN1 allow Move Command
      MRD
      LD      M2110  ; MN1 Move Command
      OR      M2745
      ANB
      OUT     M2745
      MRD
      LD      M2745
      AND     M8029  ; Instruction execution complete
      OR      M2746
      ANB
      OUT     M2746
      MPP
      AND     M2746
      MOV     K11 D2000
; Force next step after timeout
994   LD      M2152  ; Enable
      ANI     M1511  ; Communication Timeout
      AND=    K9 D2000  ; SLAVE ID SCAN H9000-H9009
      MPS
      AND     T5  ; Force next step after timeout
      MOV     K11 D2000
      MPP
      OUT     T5 K50  ; Force next step after timeout
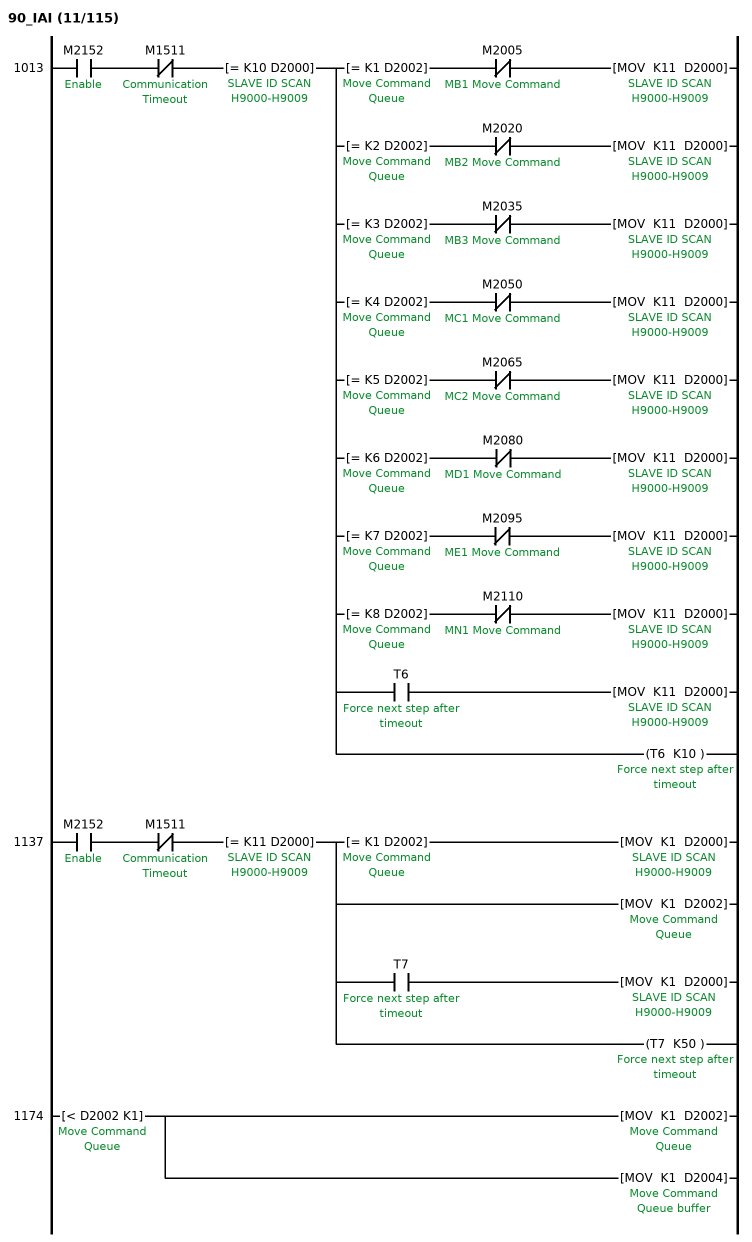
1013  LD      M2152  ; Enable
      ANI     M1511  ; Communication Timeout
      AND=    K10 D2000  ; SLAVE ID SCAN H9000-H9009
      MPS
      AND=    K1 D2002  ; Move Command Queue
      ANI     M2005  ; MB1 Move Command
      MOV     K11 D2000
      MRD
      AND=    K2 D2002  ; Move Command Queue
      ANI     M2020  ; MB2 Move Command
      MOV     K11 D2000
      MRD
      AND=    K3 D2002  ; Move Command Queue
      ANI     M2035  ; MB3 Move Command
      MOV     K11 D2000
      MRD
      AND=    K4 D2002  ; Move Command Queue
      ANI     M2050  ; MC1 Move Command
      MOV     K11 D2000
      MRD
      AND=    K5 D2002  ; Move Command Queue
      ANI     M2065  ; MC2 Move Command
      MOV     K11 D2000
      MRD
      AND=    K6 D2002  ; Move Command Queue
      ANI     M2080  ; MD1 Move Command
      MOV     K11 D2000
      MRD
      AND=    K7 D2002  ; Move Command Queue
      ANI     M2095  ; ME1 Move Command
      MOV     K11 D2000
      MRD
      AND=    K8 D2002  ; Move Command Queue
      ANI     M2110  ; MN1 Move Command
      MOV     K11 D2000
      MRD
      AND     T6  ; Force next step after timeout
      MOV     K11 D2000
      MPP
      OUT     T6 K10  ; Force next step after timeout
        [note] Force next step after timeout
1137  LD      M2152  ; Enable
      ANI     M1511  ; Communication Timeout
      AND=    K11 D2000  ; SLAVE ID SCAN H9000-H9009
      MPS
      AND=    K1 D2002  ; Move Command Queue
      MOV     K1 D2000
      MPP
      MOV     K1 D2002
      MPS
      AND     T7  ; Force next step after timeout
      MOV     K1 D2000
      MPP
      OUT     T7 K50  ; Force next step after timeout
        [note] Force next step after timeout
1174  LD<     D2002 K1  ; Move Command Queue
      MOV     K1 D2002
      MOV     K1 D2004  ; Move Command Queue buffer
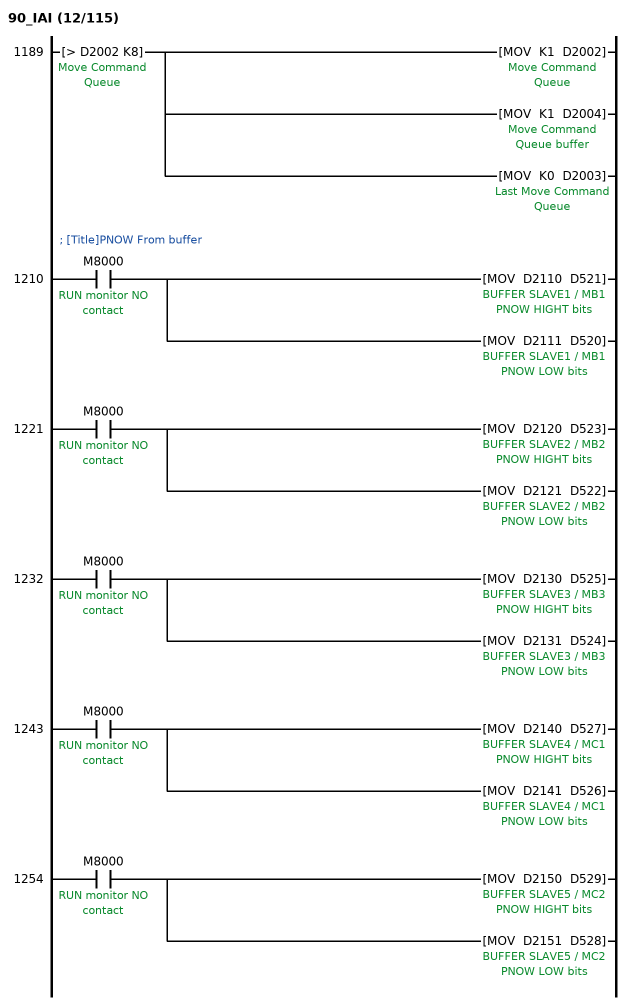
1189  LD>     D2002 K8  ; Move Command Queue
      MOV     K1 D2002
      MOV     K1 D2004
      MOV     K0 D2003
; [Title]PNOW From buffer
1210  LD      M8000  ; RUN monitor NO contact
      MOV     D2110 D521  ; MB1 PNOW HIGHT bits
      MOV     D2111 D520  ; BUFFER SLAVE1 / MB1 PNOW LOW bits
1221  LD      M8000  ; RUN monitor NO contact
      MOV     D2120 D523  ; MB2 PNOW HIGHT bits
      MOV     D2121 D522  ; BUFFER SLAVE2 / MB2 PNOW LOW bits
1232  LD      M8000  ; RUN monitor NO contact
      MOV     D2130 D525  ; MB3 PNOW HIGHT bits
      MOV     D2131 D524  ; BUFFER SLAVE3 / MB3 PNOW LOW bits
1243  LD      M8000  ; RUN monitor NO contact
      MOV     D2140 D527  ; MC1 PNOW HIGHT bits
      MOV     D2141 D526  ; BUFFER SLAVE4 / MC1 PNOW LOW bits
1254  LD      M8000  ; RUN monitor NO contact
      MOV     D2150 D529  ; MC2 PNOW HIGHT bits
      MOV     D2151 D528  ; BUFFER SLAVE5 / MC2 PNOW LOW bits
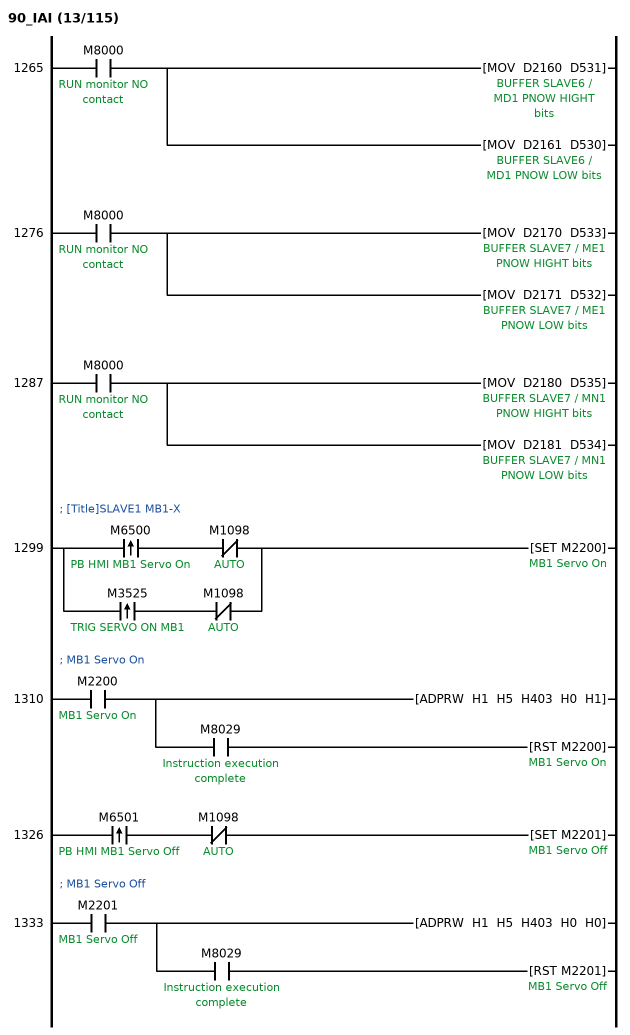
1265  LD      M8000  ; RUN monitor NO contact
      MOV     D2160 D531  ; MD1 PNOW HIGHT bits
      MOV     D2161 D530  ; BUFFER SLAVE6 / MD1 PNOW LOW bits
1276  LD      M8000  ; RUN monitor NO contact
      MOV     D2170 D533  ; ME1 PNOW HIGHT bits
      MOV     D2171 D532  ; BUFFER SLAVE7 / ME1 PNOW LOW bits
1287  LD      M8000  ; RUN monitor NO contact
      MOV     D2180 D535  ; MN1 PNOW HIGHT bits
      MOV     D2181 D534  ; BUFFER SLAVE7 / MN1 PNOW LOW bits
; [Title]SLAVE1 MB1-X
1299  LDP     M6500  ; PB HMI MB1 Servo On
      ANI     M1098  ; AUTO
      LDP     M3525  ; TRIG SERVO ON MB1
      ANI     M1098  ; AUTO
      ORB
      SET     M2200  ; MB1 Servo On
; MB1 Servo On
1310  LD      M2200  ; MB1 Servo On
      ADPRW   H1 H5 H403 H0 H1
      AND     M8029  ; Instruction execution complete
      RST     M2200  ; MB1 Servo On
1326  LDP     M6501  ; PB HMI MB1 Servo Off
      ANI     M1098  ; AUTO
      SET     M2201  ; MB1 Servo Off
; MB1 Servo Off
1333  LD      M2201  ; MB1 Servo Off
      ADPRW   H1 H5 H403 H0 H0
      AND     M8029  ; Instruction execution complete
      RST     M2201  ; MB1 Servo Off
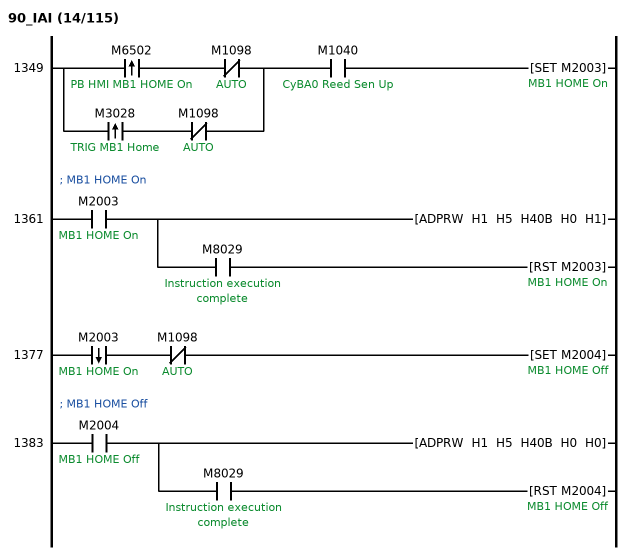
1349  LDP     M6502  ; PB HMI MB1 HOME On
      ANI     M1098  ; AUTO
      LDP     M3028  ; TRIG MB1 Home
      ANI     M1098  ; AUTO
      ORB
      AND     M1040  ; CyBA0 Reed Sen Up
      SET     M2003  ; MB1 HOME On
; MB1 HOME On
1361  LD      M2003  ; MB1 HOME On
      ADPRW   H1 H5 H40B H0 H1
      AND     M8029  ; Instruction execution complete
      RST     M2003  ; MB1 HOME On
1377  LDF     M2003  ; MB1 HOME On
      ANI     M1098  ; AUTO
      SET     M2004  ; MB1 HOME Off
; MB1 HOME Off
1383  LD      M2004  ; MB1 HOME Off
      ADPRW   H1 H5 H40B H0 H0
      AND     M8029  ; Instruction execution complete
      RST     M2004  ; MB1 HOME Off
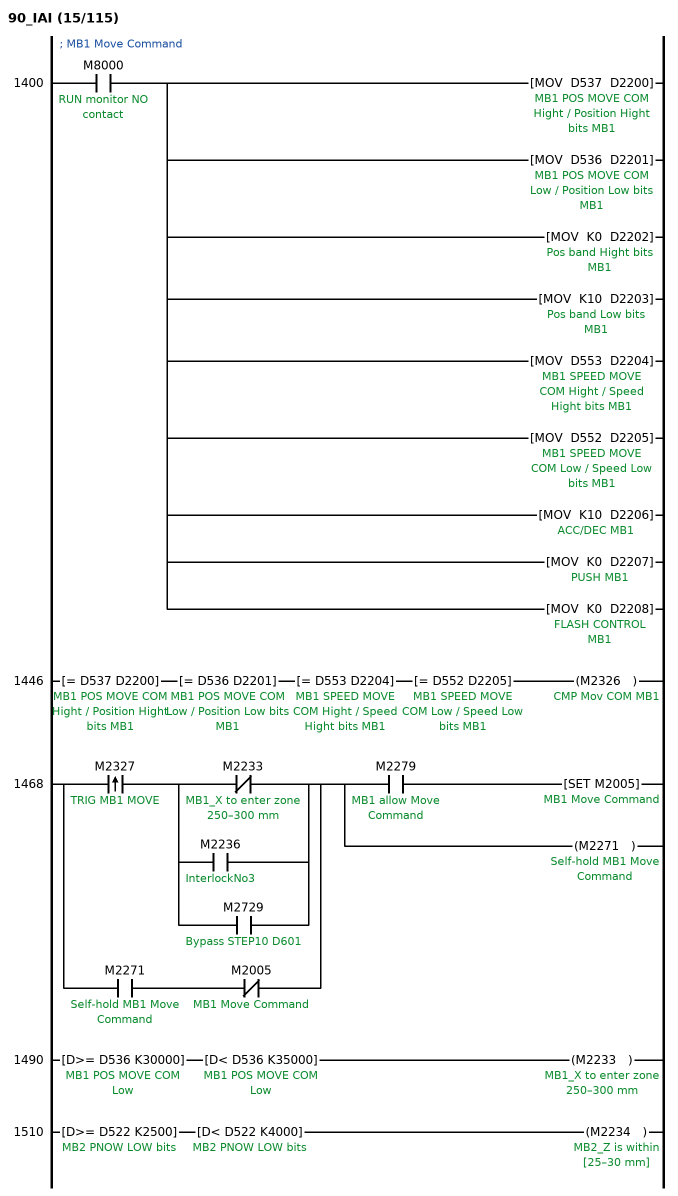
; MB1 Move Command
1400  LD      M8000  ; RUN monitor NO contact
      MOV     D537 D2200  ; MB1 POS MOVE COM Hight / Position Hight bits MB1
      MOV     D536 D2201  ; MB1 POS MOVE COM Low / Position Low bits MB1
      MOV     K0 D2202  ; Pos band Hight bits MB1
      MOV     K10 D2203  ; Pos band Low bits MB1
      MOV     D553 D2204  ; MB1 SPEED MOVE COM Hight / Speed Hight bits MB1
      MOV     D552 D2205  ; MB1 SPEED MOVE COM Low / Speed Low bits MB1
      MOV     K10 D2206  ; ACC/DEC MB1
      MOV     K0 D2207  ; PUSH MB1
      MOV     K0 D2208  ; FLASH CONTROL MB1
1446  LD=     D537 D2200  ; MB1 POS MOVE COM Hight / Position Hight bits MB1
      AND=    D536 D2201  ; MB1 POS MOVE COM Low / Position Low bits MB1
      AND=    D553 D2204  ; MB1 SPEED MOVE COM Hight / Speed Hight bits MB1
      AND=    D552 D2205  ; MB1 SPEED MOVE COM Low / Speed Low bits MB1
      OUT     M2326  ; CMP Mov COM MB1
1468  LDP     M2327  ; TRIG MB1 MOVE
      LDI     M2233  ; MB1_X to enter zone 250–300 mm
      OR      M2236  ; InterlockNo3
      OR      M2729  ; Bypass STEP10 D601
      ANB
      LD      M2271  ; Self-hold MB1 Move Command
      ANI     M2005  ; MB1 Move Command
      ORB
      MPS
      AND     M2279  ; MB1 allow Move Command
      SET     M2005  ; MB1 Move Command
      MPP
      OUT     M2271  ; Self-hold MB1 Move Command
1490  LDD>=   D536 K30000  ; MB1 POS MOVE COM Low
      ANDD<   D536 K35000  ; MB1 POS MOVE COM Low
      OUT     M2233  ; MB1_X to enter zone 250–300 mm
1510  LDD>=   D522 K2500  ; MB2 PNOW LOW bits
      ANDD<   D522 K4000  ; MB2 PNOW LOW bits
      OUT     M2234  ; MB2_Z is within [25–30 mm]
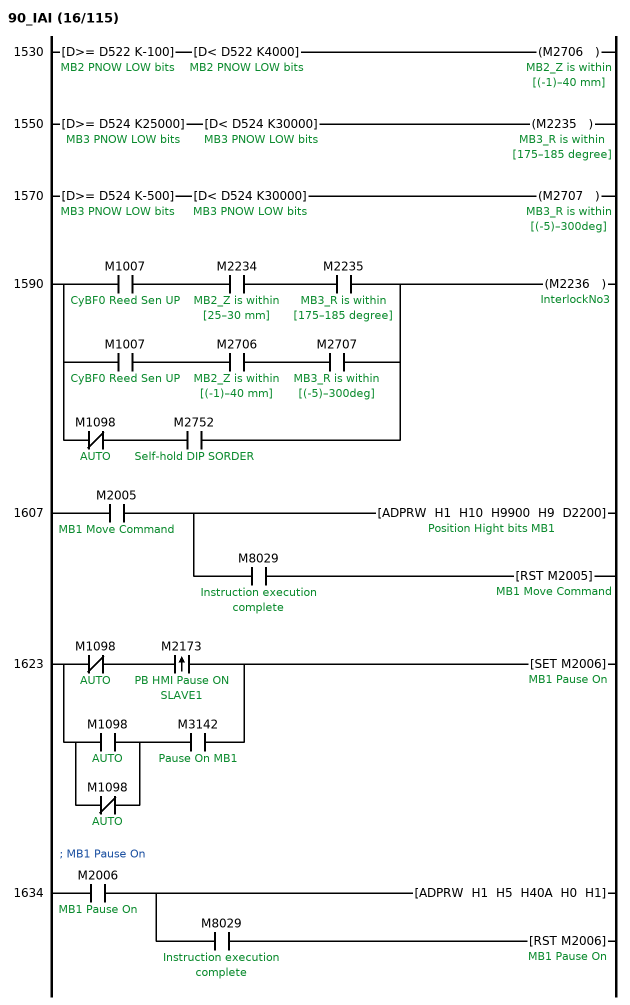
1530  LDD>=   D522 K-100  ; MB2 PNOW LOW bits
      ANDD<   D522 K4000  ; MB2 PNOW LOW bits
      OUT     M2706  ; MB2_Z is within [(-1)–40 mm]
1550  LDD>=   D524 K25000  ; MB3 PNOW LOW bits
      ANDD<   D524 K30000  ; MB3 PNOW LOW bits
      OUT     M2235  ; MB3_R is within [175–185 degree]
1570  LDD>=   D524 K-500  ; MB3 PNOW LOW bits
      ANDD<   D524 K30000  ; MB3 PNOW LOW bits
      OUT     M2707  ; MB3_R is within [(-5)–300deg]
1590  LD      M1007  ; CyBF0 Reed Sen UP
      AND     M2234  ; MB2_Z is within [25–30 mm]
      AND     M2235  ; MB3_R is within [175–185 degree]
      LD      M1007  ; CyBF0 Reed Sen UP
      AND     M2706  ; MB2_Z is within [(-1)–40 mm]
      AND     M2707  ; MB3_R is within [(-5)–300deg]
      ORB
      LDI     M1098  ; AUTO
      AND     M2752  ; Self-hold DIP SORDER
      ORB
      OUT     M2236  ; InterlockNo3
1607  LD      M2005  ; MB1 Move Command
      ADPRW   H1 H10 H9900 H9 D2200
      AND     M8029  ; Instruction execution complete
      RST     M2005  ; MB1 Move Command
1623  LDI     M1098  ; AUTO
      ANDP    M2173  ; PB HMI Pause ON SLAVE1
      LD      M1098  ; AUTO
      ORI     M1098  ; AUTO
      AND     M3142  ; Pause On MB1
      ORB
      SET     M2006  ; MB1 Pause On
; MB1 Pause On
1634  LD      M2006  ; MB1 Pause On
      ADPRW   H1 H5 H40A H0 H1
      AND     M8029  ; Instruction execution complete
      RST     M2006  ; MB1 Pause On
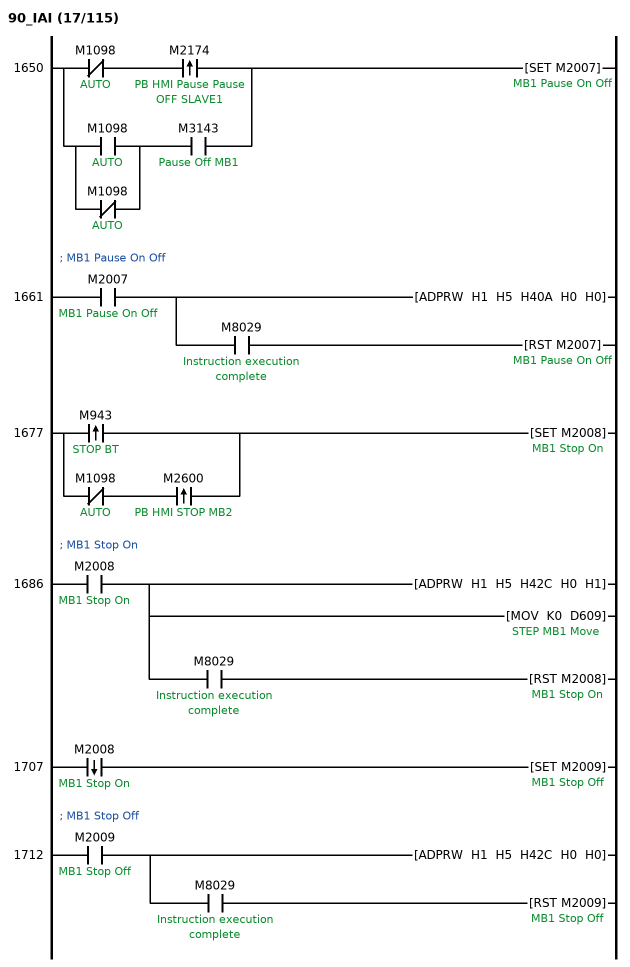
1650  LDI     M1098  ; AUTO
      ANDP    M2174  ; PB HMI Pause Pause OFF SLAVE1
      LD      M1098  ; AUTO
      ORI     M1098  ; AUTO
      AND     M3143  ; Pause Off MB1
      ORB
      SET     M2007  ; MB1 Pause On Off
; MB1 Pause On Off
1661  LD      M2007  ; MB1 Pause On Off
      ADPRW   H1 H5 H40A H0 H0
      AND     M8029  ; Instruction execution complete
      RST     M2007  ; MB1 Pause On Off
1677  LDP     M943  ; STOP BT
      LDI     M1098  ; AUTO
      ANDP    M2600  ; PB HMI STOP MB2
      ORB
      SET     M2008  ; MB1 Stop On
; MB1 Stop On
1686  LD      M2008  ; MB1 Stop On
      ADPRW   H1 H5 H42C H0 H1
      MOV     K0 D609  ; STEP MB1 Move
      AND     M8029  ; Instruction execution complete
      RST     M2008  ; MB1 Stop On
1707  LDF     M2008  ; MB1 Stop On
      SET     M2009  ; MB1 Stop Off
; MB1 Stop Off
1712  LD      M2009  ; MB1 Stop Off
      ADPRW   H1 H5 H42C H0 H0
      AND     M8029  ; Instruction execution complete
      RST     M2009  ; MB1 Stop Off
